(* CODESYS project SmiuUGP.project

Project tree, tasks and I/O mapping:
  CODESYS_Control_for_Raspberry_Pi : CODESYS Control for Raspberry Pi, 3S - Smart Software Solutions GmbH, version 3.5.7.10
    application Application
      libraries: Util, * (System); AlarmManager, * (Intern); Alarm Manager Interfaces, * (Intern); Standard, * (System); VisuDialogs, * (System)
      task MainTask (cyclic, interval t#50ms, priority 2, watchdog t#1000ms x 1) calls PLC_PRG, GPIO_HANDLER, AlarmChecker
      task VISU_TASK (cyclic, interval 100 ms, priority 30) calls VisuElems.Visu_Prg
      task AlarmManagerTask (cyclic, interval 50 ms, priority 31) calls AlarmManager.Alarm_Prg
      task BusTask (cyclic, interval t#20ms, priority 1, watchdog t#1000ms x 1) calls BusReinit
      program PLC_PRG [ST]
      image pool ImagePool
      program GPIO_HANDLER [ST]
      visualization/
        visualisation monitoring
        ups_s2/
          visualisation ups_s2_m1_state
          visualisation ups_s2_m1_params
          visualisation ups_s2
          visualisation ups_s2_m2_params
          visualisation ups_s2_m2_state
          visualisation ups_s2_m3_params
          visualisation ups_s2_m4_state
          visualisation ups_s2_m4_params
          visualisation ups_s2_m3_state
        visualisation test
        visualisation main
        visualisation info
        visualisation climate
        visualisation control
        visualisation alarm
        visualisation schrps
        visualisation shasn
        visualisation logs
        visualisation schrpa
        ups_s1/
          visualisation ups_s1
          visualisation ups_s1_m1_params
          visualisation ups_s1_m1_state
          visualisation ups_s1_m2_params
          visualisation ups_s1_m2_state
          visualisation ups_s1_m3_params
          visualisation ups_s1_m3_state
          visualisation ups_s1_m4_params
          visualisation ups_s1_m4_state
        ups_a1/
          visualisation ups_a1
          visualisation ups_a1_m1_params
          visualisation ups_a1_m1_state
          visualisation ups_a1_m2_params
          visualisation ups_a1_m2_state
        ups_a2/
          visualisation ups_a2
          visualisation ups_a2_m1_params
          visualisation ups_a2_m1_state
          visualisation ups_a2_m2_params
          visualisation ups_a2_m2_state
        visualisation climate_log
        visualisation more
      program InterviewState [ST]
      Alarm Configuration
        alarm class Error (priority 10, acknowledge REP)
        alarm class Warning (priority 30, acknowledge REP)
        alarm class Info (priority 100, acknowledge REP)
        AlarmStorage
        text list AlarmGroup
        alarm group AlarmGroup
            56 [Error]: Comparison Equal, ExpressionToCompare TRUE, Expression PLC_PRG.mpx_s2_4_alarm - "Авария ИБПС 2 модуль 4"
            46 [Error]: Comparison Equal, ExpressionToCompare TRUE, Expression PLC_PRG.mpx_a1_2_alarm - "Авария ИБПА 1 модуль 2"
            49 [Error]: Comparison Equal, ExpressionToCompare TRUE, Expression PLC_PRG.mpx_s1_1_alarm - "Авария ИБПС 1 модуль 1"
            51 [Error]: Comparison Equal, ExpressionToCompare TRUE, Expression PLC_PRG.mpx_s1_3_alarm - "Авария ИБПС 1 модуль 3"
            87 [Error]: Comparison Equal, ExpressionToCompare FALSE, Expression GPIO_HANDLER.IN_10 - "Отключен выходной автомат ИБПС 2"
            94 [Error]: Comparison Equal, ExpressionToCompare TRUE, Expression AlarmChecker.ups_a1_out_v_alarm - "Отсутствует напряжение на выходе ИБПА 1"
            54 [Error]: Comparison Equal, ExpressionToCompare TRUE, Expression PLC_PRG.mpx_s2_2_alarm - "Авария ИБПС 2 модуль 2"
            53 [Error]: Comparison Equal, ExpressionToCompare TRUE, Expression PLC_PRG.mpx_s2_1_alarm - "Авария ИБПС 2 модуль 1"
            92 [Error]: Comparison Equal, ExpressionToCompare TRUE, Expression AlarmChecker.ups_s1_out_v_alarm - "Отсутствует напряжение на выходе ИБПС 1"
            85 [Error]: Comparison Equal, ExpressionToCompare FALSE, Expression GPIO_HANDLER.IN_8 - "Отключен выходной автомат ИБПС 1"
            47 [Error]: Comparison Equal, ExpressionToCompare TRUE, Expression PLC_PRG.mpx_a2_1_alarm - "Авария ИБПА 2 модуль 1"
            90 [Error]: Comparison Equal, ExpressionToCompare TRUE, Expression AlarmChecker.ups_a1_in_v_alarm - "Отсутствует напряжение на входе ИБПА 1"
            52 [Error]: Comparison Equal, ExpressionToCompare TRUE, Expression PLC_PRG.mpx_s1_4_alarm - "Авария ИБПС 1 модуль 4"
            1 [Error]: Comparison Equal, ExpressionToCompare FALSE, Expression GPIO_HANDLER.IN_5 - "Отсутствует напряжение на резервном вводе ЩРПА"
            2 [Error]: Comparison Equal, ExpressionToCompare FALSE, Expression PLC_PRG.mv110_in_0_in_main_present - "Отсутствует напряжение на основном вводе ШАСН"
            6 [Error]: Comparison Equal, ExpressionToCompare FALSE, Expression PLC_PRG.mv110_in_2_bp_sn_present - "Отсутствует напряжение на шине БП ШАСН"
            4 [Error]: Comparison Equal, ExpressionToCompare TRUE, Expression PLC_PRG.mv110_in_7_gp1_u_fault - "Отсутствует напряжение на ГП 1 ЩРПС"
            5 [Error]: Comparison Equal, ExpressionToCompare TRUE, Expression PLC_PRG.mv110_in_8_gp2_u_fault - "Отсутствует напряжение на ГП 2 ЩРПС"
            93 [Error]: Comparison Equal, ExpressionToCompare TRUE, Expression AlarmChecker.ups_s2_out_v_alarm - "Отсутствует напряжение на выходе ИБПС 2"
            48 [Error]: Comparison Equal, ExpressionToCompare TRUE, Expression PLC_PRG.mpx_a2_2_alarm - "Авария ИБПА 2 модуль 2"
            45 [Error]: Comparison Equal, ExpressionToCompare TRUE, Expression PLC_PRG.mpx_a1_1_alarm - "Авария ИБПА 1 модуль 1"
            88 [Error]: Comparison Equal, ExpressionToCompare TRUE, Expression AlarmChecker.ups_s1_in_v_alarm - "Отсутствует напряжение на входе ИБПС 1"
            50 [Error]: Comparison Equal, ExpressionToCompare TRUE, Expression PLC_PRG.mpx_s1_2_alarm - "Авария ИБПС 1 модуль 2"
            95 [Error]: Comparison Equal, ExpressionToCompare TRUE, Expression AlarmChecker.ups_a2_out_v_alarm - "Отсутствует напряжение на выходе ИБПА 2"
            89 [Error]: Comparison Equal, ExpressionToCompare TRUE, Expression AlarmChecker.ups_s2_in_v_alarm - "Отсутствует напряжение на входе ИБПС 2"
            0 [Error]: Comparison Equal, ExpressionToCompare FALSE, Expression GPIO_HANDLER.IN_4 - "Отсутствует напряжение на основном вводе ЩРПА"
            91 [Error]: Comparison Equal, ExpressionToCompare TRUE, Expression AlarmChecker.ups_a2_in_v_alarm - "Отсутствует напряжение на входе ИБПА 2"
            55 [Error]: Comparison Equal, ExpressionToCompare TRUE, Expression PLC_PRG.mpx_s2_3_alarm - "Авария ИБПС 2 модуль 3"
            3 [Error]: Comparison Equal, ExpressionToCompare FALSE, Expression PLC_PRG.mv110_in_1_in_reserve_present - "Отсутствует напряжение на резервном вводе ШАСН"
            7 [Error]: Comparison Equal, ExpressionToCompare FALSE, Expression PLC_PRG.mv110_in_3_gp_sn_present - "Отсутствует напряжение на шине ГП ШАСН"
        text list ClimateGroup
        alarm group ClimateGroup
            1 [Info]: Comparison Equal, ExpressionToCompare TRUE, Expression PLC_PRG.climate_auto_state - "Автоматика включена"
            2 [Info]: Comparison Equal, ExpressionToCompare FALSE, Expression PLC_PRG.climate_heat_state - "Обогрев выключен"
            3 [Info]: Comparison Equal, ExpressionToCompare FALSE, Expression PLC_PRG.climate_auto_state - "Автоматика выключена"
            4 [Info]: Comparison Equal, ExpressionToCompare TRUE, Expression PLC_PRG.climate_zaslonka_state - "Заслонка открыта"
            5 [Info]: Comparison Equal, ExpressionToCompare FALSE, Expression PLC_PRG.climate_zaslonka_state - "Заслонка закрыта"
            11 [Info]: Comparison Equal, ExpressionToCompare FALSE, Expression PLC_PRG.climate_heat_door_state - "Обогрев дверей выключен"
            7 [Info]: Comparison Equal, ExpressionToCompare FALSE, Expression PLC_PRG.climate_vent_1_state - "Вентиляторы выключены"
            6 [Info]: Comparison Equal, ExpressionToCompare TRUE, Expression PLC_PRG.climate_vent_1_state - "Вентиляторы включены"
            8 [Info]: Comparison Equal, ExpressionToCompare TRUE, Expression PLC_PRG.climate_condition_1_state - "Кондиционеры включены"
            9 [Info]: Comparison Equal, ExpressionToCompare FALSE, Expression PLC_PRG.climate_condition_1_state - "Кондиционеры выключены"
            10 [Info]: Comparison Equal, ExpressionToCompare TRUE, Expression PLC_PRG.climate_heat_door_state - "Обогрев дверей включен"
            0 [Info]: Comparison Equal, ExpressionToCompare TRUE, Expression PLC_PRG.climate_heat_state - "Обогрев включен"
      program BusReinit [ST]
      program AlarmChecker [ST]
    SoftMotion General Axis Pool
    GPIOs_B_Pi2 : GPIOs B+/Pi2, 3S - Smart Software Solutions GmbH, version 1.1.1.10
        input  Application.GPIO_HANDLER.IN_10 : BOOL  // digital inputs (GPIO0..GPIO31).Bit5
        input  Application.GPIO_HANDLER.IN_12 : BOOL  // digital inputs (GPIO0..GPIO31).Bit6
        input  Application.GPIO_HANDLER.IN_9 : BOOL  // digital inputs (GPIO0..GPIO31).Bit7
        input  Application.GPIO_HANDLER.IN_8 : BOOL  // digital inputs (GPIO0..GPIO31).Bit8
        input  Application.GPIO_HANDLER.IN_3 : BOOL  // digital inputs (GPIO0..GPIO31).Bit10
        input  Application.GPIO_HANDLER.IN_11 : BOOL  // digital inputs (GPIO0..GPIO31).Bit12
        input  Application.GPIO_HANDLER.IN_1 : BOOL  // digital inputs (GPIO0..GPIO31).Bit13
        input  Application.GPIO_HANDLER.IN_6 : BOOL  // digital inputs (GPIO0..GPIO31).Bit18
        input  Application.GPIO_HANDLER.IN_7 : BOOL  // digital inputs (GPIO0..GPIO31).Bit21
        input  Application.GPIO_HANDLER.IN_5 : BOOL  // digital inputs (GPIO0..GPIO31).Bit23
        input  Application.GPIO_HANDLER.IN_4 : BOOL  // digital inputs (GPIO0..GPIO31).Bit24
        input  Application.GPIO_HANDLER.IN_2 : BOOL  // digital inputs (GPIO0..GPIO31).Bit25
        unmapped channels: digital inputs (GPIO0..GPIO31), digital outputs (GPIO0..GPIO31)
    Camera device
      <Empty>
    I²C
    SPI
    Onewire
    Ethernet : Ethernet, 3S - Smart Software Solutions GmbH, version 3.4.2.0
        settings: IPAddress = [192,168,10,200]; SubnetMask = [255,255,255,0]; GatewayAddress = [0,0,0,0]; NetworkInterfaceName = 'eth0'; NetworkInterfaceName = "eth0"
      Modbus_TCP_Master : Modbus TCP Master, 3S - Smart Software Solutions GmbH, version 3.5.4.0
          settings: AutoReconnect = TRUE
        MPX_S2_1 : Modbus TCP Slave, 3S - Smart Software Solutions GmbH, version 3.5.4.0
            settings: Unit-ID = 1; ResponseTimeout = 1500; IPAddress = [192, 168, 10, 108]; bypass_out.Function Code = 3; bypass_out.Read Offset = 16#0015; bypass_out.Read Length = 7; bypass_out.Write Offset = 0; bypass_out.Write Length = 0; bypass_out.Cycle Time = 300; output.Function Code = 3; output.Read Offset = 16#001F; output.Read Length = 13; output.Write Offset = 0; output.Write Length = 0; output.Cycle Time = 300; battery.Function Code = 3; battery.Read Offset = 16#002F; battery.Read Length = 7; battery.Write Offset = 0; battery.Write Length = 0; battery.Cycle Time = 300; states.Function Code = 3; states.Read Offset = 16#0000; states.Read Length = 2; states.Write Offset = 0; states.Write Length = 0; states.Cycle Time = 300; input.Function Code = 3; input.Read Offset = 16#000B; input.Read Length = 7; input.Write Offset = 0; input.Write Length = 0; input.Cycle Time = 300; temp.Function Code = 3; temp.Read Offset = 16#003D; temp.Read Length = 1; temp.Write Offset = 0; temp.Write Length = 0; temp.Cycle Time = 300; battery_test.Function Code = 6;
              battery_test.Read Offset = 0; battery_test.Read Length = 0; battery_test.Write Offset = 16#0070; battery_test.Write Length = 1; battery_test.Cycle Time = 100
            input  Application.PLC_PRG.mpx_s2_1_bypass_v_1 : WORD  // bypass_out.bypass_out
            input  Application.PLC_PRG.mpx_s2_1_bypass_v_2 : WORD  // bypass_out.bypass_out
            input  Application.PLC_PRG.mpx_s2_1_bypass_v_3 : WORD  // bypass_out.bypass_out
            input  Application.PLC_PRG.mpx_s2_1_bypass_freq : WORD  // bypass_out.bypass_out
            input  Application.PLC_PRG.mpx_s2_1_output_v_1 : WORD  // bypass_out.bypass_out
            input  Application.PLC_PRG.mpx_s2_1_output_v_2 : WORD  // bypass_out.bypass_out
            input  Application.PLC_PRG.mpx_s2_1_output_v_3 : WORD  // bypass_out.bypass_out
            input  Application.PLC_PRG.mpx_s2_1_output_i_1 : WORD  // output.output
            input  Application.PLC_PRG.mpx_s2_1_output_i_2 : WORD  // output.output
            input  Application.PLC_PRG.mpx_s2_1_output_i_3 : WORD  // output.output
            input  Application.PLC_PRG.mpx_s2_1_load_ph_1 : WORD  // output.output
            input  Application.PLC_PRG.mpx_s2_1_load_ph_2 : WORD  // output.output
            input  Application.PLC_PRG.mpx_s2_1_load_ph_3 : WORD  // output.output
            input  Application.PLC_PRG.mpx_s2_1_output_active_power_1 : WORD  // output.output
            input  Application.PLC_PRG.mpx_s2_1_output_active_power_2 : WORD  // output.output
            input  Application.PLC_PRG.mpx_s2_1_output_active_power_3 : WORD  // output.output
            input  Application.PLC_PRG.mpx_s2_1_output_freq : WORD  // output.output
            input  Application.PLC_PRG.mpx_s2_1_battery_voltage : WORD  // battery.battery
            input  Application.PLC_PRG.mpx_s2_1_battery_current : WORD  // battery.battery
            input  Application.PLC_PRG.mpx_s2_1_battery_capacity : WORD  // battery.battery
            input  Application.PLC_PRG.mpx_s2_1_battery_time : WORD  // battery.battery
            input  Application.PLC_PRG.mpx_s2_1_state_reg_1 : WORD  // states.states
            input  Application.PLC_PRG.mpx_s2_1_state_reg_2 : WORD  // states.states
            input  Application.PLC_PRG.mpx_s2_1_in_v_1 : WORD  // input.input
            input  Application.PLC_PRG.mpx_s2_1_in_v_2 : WORD  // input.input
            input  Application.PLC_PRG.mpx_s2_1_in_v_3 : WORD  // input.input
            input  Application.PLC_PRG.mpx_s2_1_in_freq : WORD  // input.input
            input  Application.PLC_PRG.mpx_s2_1_temp : WORD  // temp.temp
            output Application.PLC_PRG.mpx_s2_test_battery_start : BIT  // battery_test
            output Application.PLC_PRG.mpx_test_battery_command : ARRAY[0..0] OF WORD  // battery_test
            unmapped channels: bypass_out, output, battery, states, input, temp
        MPX_S2_4 : Modbus TCP Slave, 3S - Smart Software Solutions GmbH, version 3.5.4.0
            settings: Unit-ID = 1; ResponseTimeout = 1500; IPAddress = [192, 168, 10, 105]; bypass_out.Function Code = 3; bypass_out.Read Offset = 16#0015; bypass_out.Read Length = 7; bypass_out.Write Offset = 0; bypass_out.Write Length = 0; bypass_out.Cycle Time = 300; output.Function Code = 3; output.Read Offset = 16#001F; output.Read Length = 13; output.Write Offset = 0; output.Write Length = 0; output.Cycle Time = 300; battery.Function Code = 3; battery.Read Offset = 16#002F; battery.Read Length = 7; battery.Write Offset = 0; battery.Write Length = 0; battery.Cycle Time = 300; states.Function Code = 3; states.Read Offset = 16#0000; states.Read Length = 2; states.Write Offset = 0; states.Write Length = 0; states.Cycle Time = 300; input.Function Code = 3; input.Read Offset = 16#000B; input.Read Length = 7; input.Write Offset = 0; input.Write Length = 0; input.Cycle Time = 300; temp.Function Code = 3; temp.Read Offset = 16#003D; temp.Read Length = 1; temp.Write Offset = 0; temp.Write Length = 0; temp.Cycle Time = 300; battery_test.Function Code = 6;
              battery_test.Read Offset = 0; battery_test.Read Length = 0; battery_test.Write Offset = 16#0070; battery_test.Write Length = 1; battery_test.Cycle Time = 100
            input  Application.PLC_PRG.mpx_s2_4_bypass_v_1 : WORD  // bypass_out.bypass_out
            input  Application.PLC_PRG.mpx_s2_4_bypass_v_2 : WORD  // bypass_out.bypass_out
            input  Application.PLC_PRG.mpx_s2_4_bypass_v_3 : WORD  // bypass_out.bypass_out
            input  Application.PLC_PRG.mpx_s2_4_bypass_freq : WORD  // bypass_out.bypass_out
            input  Application.PLC_PRG.mpx_s2_4_output_v_1 : WORD  // bypass_out.bypass_out
            input  Application.PLC_PRG.mpx_s2_4_output_v_2 : WORD  // bypass_out.bypass_out
            input  Application.PLC_PRG.mpx_s2_4_output_v_3 : WORD  // bypass_out.bypass_out
            input  Application.PLC_PRG.mpx_s2_4_output_i_1 : WORD  // output.output
            input  Application.PLC_PRG.mpx_s2_4_output_i_2 : WORD  // output.output
            input  Application.PLC_PRG.mpx_s2_4_output_i_3 : WORD  // output.output
            input  Application.PLC_PRG.mpx_s2_4_load_ph_1 : WORD  // output.output
            input  Application.PLC_PRG.mpx_s2_4_load_ph_2 : WORD  // output.output
            input  Application.PLC_PRG.mpx_s2_4_load_ph_3 : WORD  // output.output
            input  Application.PLC_PRG.mpx_s2_4_output_active_power_1 : WORD  // output.output
            input  Application.PLC_PRG.mpx_s2_4_output_active_power_2 : WORD  // output.output
            input  Application.PLC_PRG.mpx_s2_4_output_active_power_3 : WORD  // output.output
            input  Application.PLC_PRG.mpx_s2_4_output_freq : WORD  // output.output
            input  Application.PLC_PRG.mpx_s2_4_battery_voltage : WORD  // battery.battery
            input  Application.PLC_PRG.mpx_s2_4_battery_current : WORD  // battery.battery
            input  Application.PLC_PRG.mpx_s2_4_battery_capacity : WORD  // battery.battery
            input  Application.PLC_PRG.mpx_s2_4_battery_time : WORD  // battery.battery
            input  Application.PLC_PRG.mpx_s2_4_state_reg_1 : WORD  // states.states
            input  Application.PLC_PRG.mpx_s2_4_state_reg_2 : WORD  // states.states
            input  Application.PLC_PRG.mpx_s2_4_in_v_1 : WORD  // input.input
            input  Application.PLC_PRG.mpx_s2_4_in_v_2 : WORD  // input.input
            input  Application.PLC_PRG.mpx_s2_4_in_v_3 : WORD  // input.input
            input  Application.PLC_PRG.mpx_s2_4_in_freq : WORD  // input.input
            input  Application.PLC_PRG.mpx_s2_4_temp : WORD  // temp.temp
            output Application.PLC_PRG.mpx_s2_test_battery_start : BIT  // battery_test
            output Application.PLC_PRG.mpx_test_battery_command : ARRAY[0..0] OF WORD  // battery_test
            unmapped channels: bypass_out, output, battery, states, input, temp
        MPX_S2_3 : Modbus TCP Slave, 3S - Smart Software Solutions GmbH, version 3.5.4.0
            settings: Unit-ID = 1; ResponseTimeout = 1500; IPAddress = [192, 168, 10, 106]; bypass_out.Function Code = 3; bypass_out.Read Offset = 16#0015; bypass_out.Read Length = 7; bypass_out.Write Offset = 0; bypass_out.Write Length = 0; bypass_out.Cycle Time = 300; output.Function Code = 3; output.Read Offset = 16#001F; output.Read Length = 13; output.Write Offset = 0; output.Write Length = 0; output.Cycle Time = 300; battery.Function Code = 3; battery.Read Offset = 16#002F; battery.Read Length = 7; battery.Write Offset = 0; battery.Write Length = 0; battery.Cycle Time = 300; states.Function Code = 3; states.Read Offset = 16#0000; states.Read Length = 2; states.Write Offset = 0; states.Write Length = 0; states.Cycle Time = 300; input.Function Code = 3; input.Read Offset = 16#000B; input.Read Length = 7; input.Write Offset = 0; input.Write Length = 0; input.Cycle Time = 300; temp.Function Code = 3; temp.Read Offset = 16#003D; temp.Read Length = 1; temp.Write Offset = 0; temp.Write Length = 0; temp.Cycle Time = 300; battery_test.Function Code = 6;
              battery_test.Read Offset = 0; battery_test.Read Length = 0; battery_test.Write Offset = 16#0070; battery_test.Write Length = 1; battery_test.Cycle Time = 100
            input  Application.PLC_PRG.mpx_s2_3_bypass_v_1 : WORD  // bypass_out.bypass_out
            input  Application.PLC_PRG.mpx_s2_3_bypass_v_2 : WORD  // bypass_out.bypass_out
            input  Application.PLC_PRG.mpx_s2_3_bypass_v_3 : WORD  // bypass_out.bypass_out
            input  Application.PLC_PRG.mpx_s2_3_bypass_freq : WORD  // bypass_out.bypass_out
            input  Application.PLC_PRG.mpx_s2_3_output_v_1 : WORD  // bypass_out.bypass_out
            input  Application.PLC_PRG.mpx_s2_3_output_v_2 : WORD  // bypass_out.bypass_out
            input  Application.PLC_PRG.mpx_s2_3_output_v_3 : WORD  // bypass_out.bypass_out
            input  Application.PLC_PRG.mpx_s2_3_output_i_1 : WORD  // output.output
            input  Application.PLC_PRG.mpx_s2_3_output_i_2 : WORD  // output.output
            input  Application.PLC_PRG.mpx_s2_3_output_i_3 : WORD  // output.output
            input  Application.PLC_PRG.mpx_s2_3_load_ph_1 : WORD  // output.output
            input  Application.PLC_PRG.mpx_s2_3_load_ph_2 : WORD  // output.output
            input  Application.PLC_PRG.mpx_s2_3_load_ph_3 : WORD  // output.output
            input  Application.PLC_PRG.mpx_s2_3_output_active_power_1 : WORD  // output.output
            input  Application.PLC_PRG.mpx_s2_3_output_active_power_2 : WORD  // output.output
            input  Application.PLC_PRG.mpx_s2_3_output_active_power_3 : WORD  // output.output
            input  Application.PLC_PRG.mpx_s2_3_output_freq : WORD  // output.output
            input  Application.PLC_PRG.mpx_s2_3_battery_voltage : WORD  // battery.battery
            input  Application.PLC_PRG.mpx_s2_3_battery_current : WORD  // battery.battery
            input  Application.PLC_PRG.mpx_s2_3_battery_capacity : WORD  // battery.battery
            input  Application.PLC_PRG.mpx_s2_3_battery_time : WORD  // battery.battery
            input  Application.PLC_PRG.mpx_s2_3_state_reg_1 : WORD  // states.states
            input  Application.PLC_PRG.mpx_s2_3_state_reg_2 : WORD  // states.states
            input  Application.PLC_PRG.mpx_s2_3_in_v_1 : WORD  // input.input
            input  Application.PLC_PRG.mpx_s2_3_in_v_2 : WORD  // input.input
            input  Application.PLC_PRG.mpx_s2_3_in_v_3 : WORD  // input.input
            input  Application.PLC_PRG.mpx_s2_3_in_freq : WORD  // input.input
            input  Application.PLC_PRG.mpx_s2_3_temp : WORD  // temp.temp
            output Application.PLC_PRG.mpx_s2_test_battery_start : BIT  // battery_test
            output Application.PLC_PRG.mpx_test_battery_command : ARRAY[0..0] OF WORD  // battery_test
            unmapped channels: bypass_out, output, battery, states, input, temp
        MPX_S2_2 : Modbus TCP Slave, 3S - Smart Software Solutions GmbH, version 3.5.4.0
            settings: Unit-ID = 1; ResponseTimeout = 1500; IPAddress = [192, 168, 10, 107]; bypass_out.Function Code = 3; bypass_out.Read Offset = 16#0015; bypass_out.Read Length = 7; bypass_out.Write Offset = 0; bypass_out.Write Length = 0; bypass_out.Cycle Time = 300; output.Function Code = 3; output.Read Offset = 16#001F; output.Read Length = 13; output.Write Offset = 0; output.Write Length = 0; output.Cycle Time = 300; battery.Function Code = 3; battery.Read Offset = 16#002F; battery.Read Length = 7; battery.Write Offset = 0; battery.Write Length = 0; battery.Cycle Time = 300; states.Function Code = 3; states.Read Offset = 16#0000; states.Read Length = 2; states.Write Offset = 0; states.Write Length = 0; states.Cycle Time = 300; input.Function Code = 3; input.Read Offset = 16#000B; input.Read Length = 7; input.Write Offset = 0; input.Write Length = 0; input.Cycle Time = 300; temp.Function Code = 3; temp.Read Offset = 16#003D; temp.Read Length = 1; temp.Write Offset = 0; temp.Write Length = 0; temp.Cycle Time = 300; battery_test.Function Code = 6;
              battery_test.Read Offset = 0; battery_test.Read Length = 0; battery_test.Write Offset = 16#0070; battery_test.Write Length = 1; battery_test.Cycle Time = 100
            input  Application.PLC_PRG.mpx_s2_2_bypass_v_1 : WORD  // bypass_out.bypass_out
            input  Application.PLC_PRG.mpx_s2_2_bypass_v_2 : WORD  // bypass_out.bypass_out
            input  Application.PLC_PRG.mpx_s2_2_bypass_v_3 : WORD  // bypass_out.bypass_out
            input  Application.PLC_PRG.mpx_s2_2_bypass_freq : WORD  // bypass_out.bypass_out
            input  Application.PLC_PRG.mpx_s2_2_output_v_1 : WORD  // bypass_out.bypass_out
            input  Application.PLC_PRG.mpx_s2_2_output_v_2 : WORD  // bypass_out.bypass_out
            input  Application.PLC_PRG.mpx_s2_2_output_v_3 : WORD  // bypass_out.bypass_out
            input  Application.PLC_PRG.mpx_s2_2_output_i_1 : WORD  // output.output
            input  Application.PLC_PRG.mpx_s2_2_output_i_2 : WORD  // output.output
            input  Application.PLC_PRG.mpx_s2_2_output_i_3 : WORD  // output.output
            input  Application.PLC_PRG.mpx_s2_2_load_ph_1 : WORD  // output.output
            input  Application.PLC_PRG.mpx_s2_2_load_ph_2 : WORD  // output.output
            input  Application.PLC_PRG.mpx_s2_2_load_ph_3 : WORD  // output.output
            input  Application.PLC_PRG.mpx_s2_2_output_active_power_1 : WORD  // output.output
            input  Application.PLC_PRG.mpx_s2_2_output_active_power_2 : WORD  // output.output
            input  Application.PLC_PRG.mpx_s2_2_output_active_power_3 : WORD  // output.output
            input  Application.PLC_PRG.mpx_s2_2_output_freq : WORD  // output.output
            input  Application.PLC_PRG.mpx_s2_2_battery_voltage : WORD  // battery.battery
            input  Application.PLC_PRG.mpx_s2_2_battery_current : WORD  // battery.battery
            input  Application.PLC_PRG.mpx_s2_2_battery_capacity : WORD  // battery.battery
            input  Application.PLC_PRG.mpx_s2_2_battery_time : WORD  // battery.battery
            input  Application.PLC_PRG.mpx_s2_2_state_reg_1 : WORD  // states.states
            input  Application.PLC_PRG.mpx_s2_2_state_reg_2 : WORD  // states.states
            input  Application.PLC_PRG.mpx_s2_2_in_v_1 : WORD  // input.input
            input  Application.PLC_PRG.mpx_s2_2_in_v_2 : WORD  // input.input
            input  Application.PLC_PRG.mpx_s2_2_in_v_3 : WORD  // input.input
            input  Application.PLC_PRG.mpx_s2_2_in_freq : WORD  // input.input
            input  Application.PLC_PRG.mpx_s2_2_temp : WORD  // temp.temp
            output Application.PLC_PRG.mpx_s2_test_battery_start : BIT  // battery_test
            output Application.PLC_PRG.mpx_test_battery_command : ARRAY[0..0] OF WORD  // battery_test
            unmapped channels: bypass_out, output, battery, states, input, temp
        MPX_S1_1 : Modbus TCP Slave, 3S - Smart Software Solutions GmbH, version 3.5.4.0
            settings: Unit-ID = 1; ResponseTimeout = 1500; IPAddress = [192, 168, 10, 104]; bypass_out.Function Code = 3; bypass_out.Read Offset = 16#0015; bypass_out.Read Length = 7; bypass_out.Write Offset = 0; bypass_out.Write Length = 0; bypass_out.Cycle Time = 300; output.Function Code = 3; output.Read Offset = 16#001F; output.Read Length = 13; output.Write Offset = 0; output.Write Length = 0; output.Cycle Time = 300; battery.Function Code = 3; battery.Read Offset = 16#002F; battery.Read Length = 7; battery.Write Offset = 0; battery.Write Length = 0; battery.Cycle Time = 300; states.Function Code = 3; states.Read Offset = 16#0000; states.Read Length = 2; states.Write Offset = 0; states.Write Length = 0; states.Cycle Time = 300; input.Function Code = 3; input.Read Offset = 16#000B; input.Read Length = 7; input.Write Offset = 0; input.Write Length = 0; input.Cycle Time = 300; temp.Function Code = 3; temp.Read Offset = 16#003D; temp.Read Length = 1; temp.Write Offset = 0; temp.Write Length = 0; temp.Cycle Time = 300; battery_test.Function Code = 6;
              battery_test.Read Offset = 0; battery_test.Read Length = 0; battery_test.Write Offset = 16#0070; battery_test.Write Length = 1; battery_test.Cycle Time = 100
            input  Application.PLC_PRG.mpx_s1_1_bypass_v_1 : WORD  // bypass_out.bypass_out
            input  Application.PLC_PRG.mpx_s1_1_bypass_v_2 : WORD  // bypass_out.bypass_out
            input  Application.PLC_PRG.mpx_s1_1_bypass_v_3 : WORD  // bypass_out.bypass_out
            input  Application.PLC_PRG.mpx_s1_1_bypass_freq : WORD  // bypass_out.bypass_out
            input  Application.PLC_PRG.mpx_s1_1_output_v_1 : WORD  // bypass_out.bypass_out
            input  Application.PLC_PRG.mpx_s1_1_output_v_2 : WORD  // bypass_out.bypass_out
            input  Application.PLC_PRG.mpx_s1_1_output_v_3 : WORD  // bypass_out.bypass_out
            input  Application.PLC_PRG.mpx_s1_1_output_i_1 : WORD  // output.output
            input  Application.PLC_PRG.mpx_s1_1_output_i_2 : WORD  // output.output
            input  Application.PLC_PRG.mpx_s1_1_output_i_3 : WORD  // output.output
            input  Application.PLC_PRG.mpx_s1_1_load_ph_1 : WORD  // output.output
            input  Application.PLC_PRG.mpx_s1_1_load_ph_2 : WORD  // output.output
            input  Application.PLC_PRG.mpx_s1_1_load_ph_3 : WORD  // output.output
            input  Application.PLC_PRG.mpx_s1_1_output_active_power_1 : WORD  // output.output
            input  Application.PLC_PRG.mpx_s1_1_output_active_power_2 : WORD  // output.output
            input  Application.PLC_PRG.mpx_s1_1_output_active_power_3 : WORD  // output.output
            input  Application.PLC_PRG.mpx_s1_1_output_freq : WORD  // output.output
            input  Application.PLC_PRG.mpx_s1_1_battery_voltage : WORD  // battery.battery
            input  Application.PLC_PRG.mpx_s1_1_battery_current : WORD  // battery.battery
            input  Application.PLC_PRG.mpx_s1_1_battery_capacity : WORD  // battery.battery
            input  Application.PLC_PRG.mpx_s1_1_battery_time : WORD  // battery.battery
            input  Application.PLC_PRG.mpx_s1_1_state_reg_1 : WORD  // states.states
            input  Application.PLC_PRG.mpx_s1_1_state_reg_2 : WORD  // states.states
            input  Application.PLC_PRG.mpx_s1_1_in_v_1 : WORD  // input.input
            input  Application.PLC_PRG.mpx_s1_1_in_v_2 : WORD  // input.input
            input  Application.PLC_PRG.mpx_s1_1_in_v_3 : WORD  // input.input
            input  Application.PLC_PRG.mpx_s1_1_in_freq : WORD  // input.input
            input  Application.PLC_PRG.mpx_s1_1_temp : WORD  // temp.temp
            output Application.PLC_PRG.mpx_s1_test_battery_start : BIT  // battery_test
            output Application.PLC_PRG.mpx_test_battery_command : ARRAY[0..0] OF WORD  // battery_test
            unmapped channels: bypass_out, output, battery, states, input, temp
        MPX_S1_2 : Modbus TCP Slave, 3S - Smart Software Solutions GmbH, version 3.5.4.0
            settings: Unit-ID = 1; ResponseTimeout = 1500; IPAddress = [192, 168, 10, 103]; bypass_out.Function Code = 3; bypass_out.Read Offset = 16#0015; bypass_out.Read Length = 7; bypass_out.Write Offset = 0; bypass_out.Write Length = 0; bypass_out.Cycle Time = 300; output.Function Code = 3; output.Read Offset = 16#001F; output.Read Length = 13; output.Write Offset = 0; output.Write Length = 0; output.Cycle Time = 300; battery.Function Code = 3; battery.Read Offset = 16#002F; battery.Read Length = 7; battery.Write Offset = 0; battery.Write Length = 0; battery.Cycle Time = 300; states.Function Code = 3; states.Read Offset = 16#0000; states.Read Length = 2; states.Write Offset = 0; states.Write Length = 0; states.Cycle Time = 300; input.Function Code = 3; input.Read Offset = 16#000B; input.Read Length = 7; input.Write Offset = 0; input.Write Length = 0; input.Cycle Time = 300; temp.Function Code = 3; temp.Read Offset = 16#003D; temp.Read Length = 1; temp.Write Offset = 0; temp.Write Length = 0; temp.Cycle Time = 300; battery_test.Function Code = 6;
              battery_test.Read Offset = 0; battery_test.Read Length = 0; battery_test.Write Offset = 16#0070; battery_test.Write Length = 1; battery_test.Cycle Time = 100
            input  Application.PLC_PRG.mpx_s1_2_bypass_v_1 : WORD  // bypass_out.bypass_out
            input  Application.PLC_PRG.mpx_s1_2_bypass_v_2 : WORD  // bypass_out.bypass_out
            input  Application.PLC_PRG.mpx_s1_2_bypass_v_3 : WORD  // bypass_out.bypass_out
            input  Application.PLC_PRG.mpx_s1_2_bypass_freq : WORD  // bypass_out.bypass_out
            input  Application.PLC_PRG.mpx_s1_2_output_v_1 : WORD  // bypass_out.bypass_out
            input  Application.PLC_PRG.mpx_s1_2_output_v_2 : WORD  // bypass_out.bypass_out
            input  Application.PLC_PRG.mpx_s1_2_output_v_3 : WORD  // bypass_out.bypass_out
            input  Application.PLC_PRG.mpx_s1_2_output_i_1 : WORD  // output.output
            input  Application.PLC_PRG.mpx_s1_2_output_i_2 : WORD  // output.output
            input  Application.PLC_PRG.mpx_s1_2_output_i_3 : WORD  // output.output
            input  Application.PLC_PRG.mpx_s1_2_load_ph_1 : WORD  // output.output
            input  Application.PLC_PRG.mpx_s1_2_load_ph_2 : WORD  // output.output
            input  Application.PLC_PRG.mpx_s1_2_load_ph_3 : WORD  // output.output
            input  Application.PLC_PRG.mpx_s1_2_output_active_power_1 : WORD  // output.output
            input  Application.PLC_PRG.mpx_s1_2_output_active_power_2 : WORD  // output.output
            input  Application.PLC_PRG.mpx_s1_2_output_active_power_3 : WORD  // output.output
            input  Application.PLC_PRG.mpx_s1_2_output_freq : WORD  // output.output
            input  Application.PLC_PRG.mpx_s1_2_battery_voltage : WORD  // battery.battery
            input  Application.PLC_PRG.mpx_s1_2_battery_current : WORD  // battery.battery
            input  Application.PLC_PRG.mpx_s1_2_battery_capacity : WORD  // battery.battery
            input  Application.PLC_PRG.mpx_s1_2_battery_time : WORD  // battery.battery
            input  Application.PLC_PRG.mpx_s1_2_state_reg_1 : WORD  // states.states
            input  Application.PLC_PRG.mpx_s1_2_state_reg_2 : WORD  // states.states
            input  Application.PLC_PRG.mpx_s1_2_in_v_1 : WORD  // input.input
            input  Application.PLC_PRG.mpx_s1_2_in_v_2 : WORD  // input.input
            input  Application.PLC_PRG.mpx_s1_2_in_v_3 : WORD  // input.input
            input  Application.PLC_PRG.mpx_s1_2_in_freq : WORD  // input.input
            input  Application.PLC_PRG.mpx_s1_2_temp : WORD  // temp.temp
            output Application.PLC_PRG.mpx_s1_test_battery_start : BIT  // battery_test
            output Application.PLC_PRG.mpx_test_battery_command : ARRAY[0..0] OF WORD  // battery_test
            unmapped channels: bypass_out, output, battery, states, input, temp
        MPX_S1_3 : Modbus TCP Slave, 3S - Smart Software Solutions GmbH, version 3.5.4.0
            settings: Unit-ID = 1; ResponseTimeout = 1500; IPAddress = [192, 168, 10, 102]; bypass_out.Function Code = 3; bypass_out.Read Offset = 16#0015; bypass_out.Read Length = 7; bypass_out.Write Offset = 0; bypass_out.Write Length = 0; bypass_out.Cycle Time = 300; output.Function Code = 3; output.Read Offset = 16#001F; output.Read Length = 13; output.Write Offset = 0; output.Write Length = 0; output.Cycle Time = 300; battery.Function Code = 3; battery.Read Offset = 16#002F; battery.Read Length = 7; battery.Write Offset = 0; battery.Write Length = 0; battery.Cycle Time = 300; states.Function Code = 3; states.Read Offset = 16#0000; states.Read Length = 2; states.Write Offset = 0; states.Write Length = 0; states.Cycle Time = 300; input.Function Code = 3; input.Read Offset = 16#000B; input.Read Length = 7; input.Write Offset = 0; input.Write Length = 0; input.Cycle Time = 300; temp.Function Code = 3; temp.Read Offset = 16#003D; temp.Read Length = 1; temp.Write Offset = 0; temp.Write Length = 0; temp.Cycle Time = 300; battery_test.Function Code = 6;
              battery_test.Read Offset = 0; battery_test.Read Length = 0; battery_test.Write Offset = 16#0070; battery_test.Write Length = 1; battery_test.Cycle Time = 100
            input  Application.PLC_PRG.mpx_s1_3_bypass_v_1 : WORD  // bypass_out.bypass_out
            input  Application.PLC_PRG.mpx_s1_3_bypass_v_2 : WORD  // bypass_out.bypass_out
            input  Application.PLC_PRG.mpx_s1_3_bypass_v_3 : WORD  // bypass_out.bypass_out
            input  Application.PLC_PRG.mpx_s1_3_bypass_freq : WORD  // bypass_out.bypass_out
            input  Application.PLC_PRG.mpx_s1_3_output_v_1 : WORD  // bypass_out.bypass_out
            input  Application.PLC_PRG.mpx_s1_3_output_v_2 : WORD  // bypass_out.bypass_out
            input  Application.PLC_PRG.mpx_s1_3_output_v_3 : WORD  // bypass_out.bypass_out
            input  Application.PLC_PRG.mpx_s1_3_output_i_1 : WORD  // output.output
            input  Application.PLC_PRG.mpx_s1_3_output_i_2 : WORD  // output.output
            input  Application.PLC_PRG.mpx_s1_3_output_i_3 : WORD  // output.output
            input  Application.PLC_PRG.mpx_s1_3_load_ph_1 : WORD  // output.output
            input  Application.PLC_PRG.mpx_s1_3_load_ph_2 : WORD  // output.output
            input  Application.PLC_PRG.mpx_s1_3_load_ph_3 : WORD  // output.output
            input  Application.PLC_PRG.mpx_s1_3_output_active_power_1 : WORD  // output.output
            input  Application.PLC_PRG.mpx_s1_3_output_active_power_2 : WORD  // output.output
            input  Application.PLC_PRG.mpx_s1_3_output_active_power_3 : WORD  // output.output
            input  Application.PLC_PRG.mpx_s1_3_output_freq : WORD  // output.output
            input  Application.PLC_PRG.mpx_s1_3_battery_voltage : WORD  // battery.battery
            input  Application.PLC_PRG.mpx_s1_3_battery_current : WORD  // battery.battery
            input  Application.PLC_PRG.mpx_s1_3_battery_capacity : WORD  // battery.battery
            input  Application.PLC_PRG.mpx_s1_3_battery_time : WORD  // battery.battery
            input  Application.PLC_PRG.mpx_s1_3_state_reg_1 : WORD  // states.states
            input  Application.PLC_PRG.mpx_s1_3_state_reg_2 : WORD  // states.states
            input  Application.PLC_PRG.mpx_s1_3_in_v_1 : WORD  // input.input
            input  Application.PLC_PRG.mpx_s1_3_in_v_2 : WORD  // input.input
            input  Application.PLC_PRG.mpx_s1_3_in_v_3 : WORD  // input.input
            input  Application.PLC_PRG.mpx_s1_3_in_freq : WORD  // input.input
            input  Application.PLC_PRG.mpx_s1_3_temp : WORD  // temp.temp
            output Application.PLC_PRG.mpx_s1_test_battery_start : BIT  // battery_test
            output Application.PLC_PRG.mpx_test_battery_command : ARRAY[0..0] OF WORD  // battery_test
            unmapped channels: bypass_out, output, battery, states, input, temp
        MPX_S1_4 : Modbus TCP Slave, 3S - Smart Software Solutions GmbH, version 3.5.4.0
            settings: Unit-ID = 1; ResponseTimeout = 1500; IPAddress = [192, 168, 10, 101]; bypass_out.Function Code = 3; bypass_out.Read Offset = 16#0015; bypass_out.Read Length = 7; bypass_out.Write Offset = 0; bypass_out.Write Length = 0; bypass_out.Cycle Time = 300; output.Function Code = 3; output.Read Offset = 16#001F; output.Read Length = 13; output.Write Offset = 0; output.Write Length = 0; output.Cycle Time = 300; battery.Function Code = 3; battery.Read Offset = 16#002F; battery.Read Length = 7; battery.Write Offset = 0; battery.Write Length = 0; battery.Cycle Time = 300; states.Function Code = 3; states.Read Offset = 16#0000; states.Read Length = 2; states.Write Offset = 0; states.Write Length = 0; states.Cycle Time = 300; input.Function Code = 3; input.Read Offset = 16#000B; input.Read Length = 7; input.Write Offset = 0; input.Write Length = 0; input.Cycle Time = 300; temp.Function Code = 3; temp.Read Offset = 16#003D; temp.Read Length = 1; temp.Write Offset = 0; temp.Write Length = 0; temp.Cycle Time = 300; battery_test.Function Code = 6;
              battery_test.Read Offset = 0; battery_test.Read Length = 0; battery_test.Write Offset = 16#0070; battery_test.Write Length = 1; battery_test.Cycle Time = 100
            input  Application.PLC_PRG.mpx_s1_4_bypass_v_1 : WORD  // bypass_out.bypass_out
            input  Application.PLC_PRG.mpx_s1_4_bypass_v_2 : WORD  // bypass_out.bypass_out
            input  Application.PLC_PRG.mpx_s1_4_bypass_v_3 : WORD  // bypass_out.bypass_out
            input  Application.PLC_PRG.mpx_s1_4_bypass_freq : WORD  // bypass_out.bypass_out
            input  Application.PLC_PRG.mpx_s1_4_output_v_1 : WORD  // bypass_out.bypass_out
            input  Application.PLC_PRG.mpx_s1_4_output_v_2 : WORD  // bypass_out.bypass_out
            input  Application.PLC_PRG.mpx_s1_4_output_v_3 : WORD  // bypass_out.bypass_out
            input  Application.PLC_PRG.mpx_s1_4_output_i_1 : WORD  // output.output
            input  Application.PLC_PRG.mpx_s1_4_output_i_2 : WORD  // output.output
            input  Application.PLC_PRG.mpx_s1_4_output_i_3 : WORD  // output.output
            input  Application.PLC_PRG.mpx_s1_4_load_ph_1 : WORD  // output.output
            input  Application.PLC_PRG.mpx_s1_4_load_ph_2 : WORD  // output.output
            input  Application.PLC_PRG.mpx_s1_4_load_ph_3 : WORD  // output.output
            input  Application.PLC_PRG.mpx_s1_4_output_active_power_1 : WORD  // output.output
            input  Application.PLC_PRG.mpx_s1_4_output_active_power_2 : WORD  // output.output
            input  Application.PLC_PRG.mpx_s1_4_output_active_power_3 : WORD  // output.output
            input  Application.PLC_PRG.mpx_s1_4_output_freq : WORD  // output.output
            input  Application.PLC_PRG.mpx_s1_4_battery_voltage : WORD  // battery.battery
            input  Application.PLC_PRG.mpx_s1_4_battery_current : WORD  // battery.battery
            input  Application.PLC_PRG.mpx_s1_4_battery_capacity : WORD  // battery.battery
            input  Application.PLC_PRG.mpx_s1_4_battery_time : WORD  // battery.battery
            input  Application.PLC_PRG.mpx_s1_4_state_reg_1 : WORD  // states.states
            input  Application.PLC_PRG.mpx_s1_4_state_reg_2 : WORD  // states.states
            input  Application.PLC_PRG.mpx_s1_4_in_v_1 : WORD  // input.input
            input  Application.PLC_PRG.mpx_s1_4_in_v_2 : WORD  // input.input
            input  Application.PLC_PRG.mpx_s1_4_in_v_3 : WORD  // input.input
            input  Application.PLC_PRG.mpx_s1_4_in_freq : WORD  // input.input
            input  Application.PLC_PRG.mpx_s1_4_temp : WORD  // temp.temp
            output Application.PLC_PRG.mpx_s1_test_battery_start : BIT  // battery_test
            output Application.PLC_PRG.mpx_test_battery_command : ARRAY[0..0] OF WORD  // battery_test
            unmapped channels: bypass_out, output, battery, states, input, temp
        MPX_A1_1 : Modbus TCP Slave, 3S - Smart Software Solutions GmbH, version 3.5.4.0
            settings: Unit-ID = 1; ResponseTimeout = 1500; IPAddress = [192, 168, 10, 112]; bypass_out.Function Code = 3; bypass_out.Read Offset = 16#0015; bypass_out.Read Length = 7; bypass_out.Write Offset = 0; bypass_out.Write Length = 0; bypass_out.Cycle Time = 300; output.Function Code = 3; output.Read Offset = 16#001F; output.Read Length = 13; output.Write Offset = 0; output.Write Length = 0; output.Cycle Time = 300; battery.Function Code = 3; battery.Read Offset = 16#002F; battery.Read Length = 7; battery.Write Offset = 0; battery.Write Length = 0; battery.Cycle Time = 300; states.Function Code = 3; states.Read Offset = 16#0000; states.Read Length = 2; states.Write Offset = 0; states.Write Length = 0; states.Cycle Time = 300; input.Function Code = 3; input.Read Offset = 16#000B; input.Read Length = 7; input.Write Offset = 0; input.Write Length = 0; input.Cycle Time = 300; temp.Function Code = 3; temp.Read Offset = 16#003D; temp.Read Length = 1; temp.Write Offset = 0; temp.Write Length = 0; temp.Cycle Time = 300; battery_test.Function Code = 6;
              battery_test.Read Offset = 0; battery_test.Read Length = 0; battery_test.Write Offset = 16#0070; battery_test.Write Length = 1; battery_test.Cycle Time = 100
            input  Application.PLC_PRG.mpx_a1_1_bypass_v_1 : WORD  // bypass_out.bypass_out
            input  Application.PLC_PRG.mpx_a1_1_bypass_freq : WORD  // bypass_out.bypass_out
            input  Application.PLC_PRG.mpx_a1_1_output_v_1 : WORD  // bypass_out.bypass_out
            input  Application.PLC_PRG.mpx_a1_1_output_i_1 : WORD  // output.output
            input  Application.PLC_PRG.mpx_a1_1_load_ph_1 : WORD  // output.output
            input  Application.PLC_PRG.mpx_a1_1_output_active_power_1 : WORD  // output.output
            input  Application.PLC_PRG.mpx_a1_1_output_freq : WORD  // output.output
            input  Application.PLC_PRG.mpx_a1_1_battery_voltage : WORD  // battery.battery
            input  Application.PLC_PRG.mpx_a1_1_battery_current : WORD  // battery.battery
            input  Application.PLC_PRG.mpx_a1_1_battery_capacity : WORD  // battery.battery
            input  Application.PLC_PRG.mpx_a1_1_battery_time : WORD  // battery.battery
            input  Application.PLC_PRG.mpx_a1_1_state_reg_1 : WORD  // states.states
            input  Application.PLC_PRG.mpx_a1_1_state_reg_2 : WORD  // states.states
            input  Application.PLC_PRG.mpx_a1_1_in_v_1 : WORD  // input.input
            input  Application.PLC_PRG.mpx_a1_1_in_v_2 : WORD  // input.input
            input  Application.PLC_PRG.mpx_a1_1_in_v_3 : WORD  // input.input
            input  Application.PLC_PRG.mpx_a1_1_in_freq : WORD  // input.input
            input  Application.PLC_PRG.mpx_a1_1_temp : WORD  // temp.temp
            output Application.PLC_PRG.mpx_a1_test_battery_start : BIT  // battery_test
            output Application.PLC_PRG.mpx_test_battery_command : ARRAY[0..0] OF WORD  // battery_test
            unmapped channels: bypass_out, output, battery, states, input, temp
        MPX_A1_2 : Modbus TCP Slave, 3S - Smart Software Solutions GmbH, version 3.5.4.0
            settings: Unit-ID = 1; ResponseTimeout = 1500; IPAddress = [192, 168, 10, 111]; bypass_out.Function Code = 3; bypass_out.Read Offset = 16#0015; bypass_out.Read Length = 7; bypass_out.Write Offset = 0; bypass_out.Write Length = 0; bypass_out.Cycle Time = 300; output.Function Code = 3; output.Read Offset = 16#001F; output.Read Length = 13; output.Write Offset = 0; output.Write Length = 0; output.Cycle Time = 300; battery.Function Code = 3; battery.Read Offset = 16#002F; battery.Read Length = 7; battery.Write Offset = 0; battery.Write Length = 0; battery.Cycle Time = 300; states.Function Code = 3; states.Read Offset = 16#0000; states.Read Length = 2; states.Write Offset = 0; states.Write Length = 0; states.Cycle Time = 300; input.Function Code = 3; input.Read Offset = 16#000B; input.Read Length = 7; input.Write Offset = 0; input.Write Length = 0; input.Cycle Time = 300; temp.Function Code = 3; temp.Read Offset = 16#003D; temp.Read Length = 1; temp.Write Offset = 0; temp.Write Length = 0; temp.Cycle Time = 300; battery_test.Function Code = 6;
              battery_test.Read Offset = 0; battery_test.Read Length = 0; battery_test.Write Offset = 16#0070; battery_test.Write Length = 1; battery_test.Cycle Time = 100
            input  Application.PLC_PRG.mpx_a1_2_bypass_v_1 : WORD  // bypass_out.bypass_out
            input  Application.PLC_PRG.mpx_a1_2_bypass_v_2 : WORD  // bypass_out.bypass_out
            input  Application.PLC_PRG.mpx_a1_2_bypass_v_3 : WORD  // bypass_out.bypass_out
            input  Application.PLC_PRG.mpx_a1_2_bypass_freq : WORD  // bypass_out.bypass_out
            input  Application.PLC_PRG.mpx_a1_2_output_v_1 : WORD  // bypass_out.bypass_out
            input  Application.PLC_PRG.mpx_a1_2_output_v_2 : WORD  // bypass_out.bypass_out
            input  Application.PLC_PRG.mpx_a1_2_output_v_3 : WORD  // bypass_out.bypass_out
            input  Application.PLC_PRG.mpx_a1_2_output_i_1 : WORD  // output.output
            input  Application.PLC_PRG.mpx_a1_2_output_i_2 : WORD  // output.output
            input  Application.PLC_PRG.mpx_a1_2_output_i_3 : WORD  // output.output
            input  Application.PLC_PRG.mpx_a1_2_load_ph_1 : WORD  // output.output
            input  Application.PLC_PRG.mpx_a1_2_load_ph_2 : WORD  // output.output
            input  Application.PLC_PRG.mpx_a1_2_load_ph_3 : WORD  // output.output
            input  Application.PLC_PRG.mpx_a1_2_output_active_power_1 : WORD  // output.output
            input  Application.PLC_PRG.mpx_a1_2_output_active_power_2 : WORD  // output.output
            input  Application.PLC_PRG.mpx_a1_2_output_active_power_3 : WORD  // output.output
            input  Application.PLC_PRG.mpx_a1_2_output_freq : WORD  // output.output
            input  Application.PLC_PRG.mpx_a1_2_battery_voltage : WORD  // battery.battery
            input  Application.PLC_PRG.mpx_a1_2_battery_current : WORD  // battery.battery
            input  Application.PLC_PRG.mpx_a1_2_battery_capacity : WORD  // battery.battery
            input  Application.PLC_PRG.mpx_a1_2_battery_time : WORD  // battery.battery
            input  Application.PLC_PRG.mpx_a1_2_state_reg_1 : WORD  // states.states
            input  Application.PLC_PRG.mpx_a1_2_state_reg_2 : WORD  // states.states
            input  Application.PLC_PRG.mpx_a1_2_in_v_1 : WORD  // input.input
            input  Application.PLC_PRG.mpx_a1_2_in_v_2 : WORD  // input.input
            input  Application.PLC_PRG.mpx_a1_2_in_v_3 : WORD  // input.input
            input  Application.PLC_PRG.mpx_a1_2_in_freq : WORD  // input.input
            input  Application.PLC_PRG.mpx_a1_2_temp : WORD  // temp.temp
            output Application.PLC_PRG.mpx_a1_test_battery_start : BIT  // battery_test
            output Application.PLC_PRG.mpx_test_battery_command : ARRAY[0..0] OF WORD  // battery_test
            unmapped channels: bypass_out, output, battery, states, input, temp
        MPX_A2_2 : Modbus TCP Slave, 3S - Smart Software Solutions GmbH, version 3.5.4.0
            settings: Unit-ID = 1; ResponseTimeout = 1500; IPAddress = [192, 168, 10, 109]; bypass_out.Function Code = 3; bypass_out.Read Offset = 16#0015; bypass_out.Read Length = 7; bypass_out.Write Offset = 0; bypass_out.Write Length = 0; bypass_out.Cycle Time = 300; output.Function Code = 3; output.Read Offset = 16#001F; output.Read Length = 13; output.Write Offset = 0; output.Write Length = 0; output.Cycle Time = 300; battery.Function Code = 3; battery.Read Offset = 16#002F; battery.Read Length = 7; battery.Write Offset = 0; battery.Write Length = 0; battery.Cycle Time = 300; states.Function Code = 3; states.Read Offset = 16#0000; states.Read Length = 2; states.Write Offset = 0; states.Write Length = 0; states.Cycle Time = 300; input.Function Code = 3; input.Read Offset = 16#000B; input.Read Length = 7; input.Write Offset = 0; input.Write Length = 0; input.Cycle Time = 300; temp.Function Code = 3; temp.Read Offset = 16#003D; temp.Read Length = 1; temp.Write Offset = 0; temp.Write Length = 0; temp.Cycle Time = 300; battery_test.Function Code = 6;
              battery_test.Read Offset = 0; battery_test.Read Length = 0; battery_test.Write Offset = 16#0070; battery_test.Write Length = 1; battery_test.Cycle Time = 100
            input  Application.PLC_PRG.mpx_a2_2_bypass_v_1 : WORD  // bypass_out.bypass_out
            input  Application.PLC_PRG.mpx_a2_2_bypass_v_2 : WORD  // bypass_out.bypass_out
            input  Application.PLC_PRG.mpx_a2_2_bypass_v_3 : WORD  // bypass_out.bypass_out
            input  Application.PLC_PRG.mpx_a2_2_bypass_freq : WORD  // bypass_out.bypass_out
            input  Application.PLC_PRG.mpx_a2_2_output_v_1 : WORD  // bypass_out.bypass_out
            input  Application.PLC_PRG.mpx_a2_2_output_v_2 : WORD  // bypass_out.bypass_out
            input  Application.PLC_PRG.mpx_a2_2_output_v_3 : WORD  // bypass_out.bypass_out
            input  Application.PLC_PRG.mpx_a2_2_output_i_1 : WORD  // output.output
            input  Application.PLC_PRG.mpx_a2_2_output_i_2 : WORD  // output.output
            input  Application.PLC_PRG.mpx_a2_2_output_i_3 : WORD  // output.output
            input  Application.PLC_PRG.mpx_a2_2_load_ph_1 : WORD  // output.output
            input  Application.PLC_PRG.mpx_a2_2_load_ph_2 : WORD  // output.output
            input  Application.PLC_PRG.mpx_a2_2_load_ph_3 : WORD  // output.output
            input  Application.PLC_PRG.mpx_a2_2_output_active_power_1 : WORD  // output.output
            input  Application.PLC_PRG.mpx_a2_2_output_active_power_2 : WORD  // output.output
            input  Application.PLC_PRG.mpx_a2_2_output_active_power_3 : WORD  // output.output
            input  Application.PLC_PRG.mpx_a2_2_output_freq : WORD  // output.output
            input  Application.PLC_PRG.mpx_a2_2_battery_voltage : WORD  // battery.battery
            input  Application.PLC_PRG.mpx_a2_2_battery_current : WORD  // battery.battery
            input  Application.PLC_PRG.mpx_a2_2_battery_capacity : WORD  // battery.battery
            input  Application.PLC_PRG.mpx_a2_2_battery_time : WORD  // battery.battery
            input  Application.PLC_PRG.mpx_a2_2_state_reg_1 : WORD  // states.states
            input  Application.PLC_PRG.mpx_a2_2_state_reg_2 : WORD  // states.states
            input  Application.PLC_PRG.mpx_a2_2_in_v_1 : WORD  // input.input
            input  Application.PLC_PRG.mpx_a2_2_in_v_2 : WORD  // input.input
            input  Application.PLC_PRG.mpx_a2_2_in_v_3 : WORD  // input.input
            input  Application.PLC_PRG.mpx_a2_2_in_freq : WORD  // input.input
            input  Application.PLC_PRG.mpx_a2_2_temp : WORD  // temp.temp
            output Application.PLC_PRG.mpx_a2_test_battery_start : BIT  // battery_test
            output Application.PLC_PRG.mpx_test_battery_command : ARRAY[0..0] OF WORD  // battery_test
            unmapped channels: bypass_out, output, battery, states, input, temp
        MPX_A2_1 : Modbus TCP Slave, 3S - Smart Software Solutions GmbH, version 3.5.4.0
            settings: Unit-ID = 1; ResponseTimeout = 1500; IPAddress = [192, 168, 10, 110]; bypass_out.Function Code = 3; bypass_out.Read Offset = 16#0015; bypass_out.Read Length = 7; bypass_out.Write Offset = 0; bypass_out.Write Length = 0; bypass_out.Cycle Time = 300; output.Function Code = 3; output.Read Offset = 16#001F; output.Read Length = 13; output.Write Offset = 0; output.Write Length = 0; output.Cycle Time = 300; battery.Function Code = 3; battery.Read Offset = 16#002F; battery.Read Length = 7; battery.Write Offset = 0; battery.Write Length = 0; battery.Cycle Time = 300; states.Function Code = 3; states.Read Offset = 16#0000; states.Read Length = 2; states.Write Offset = 0; states.Write Length = 0; states.Cycle Time = 300; input.Function Code = 3; input.Read Offset = 16#000B; input.Read Length = 7; input.Write Offset = 0; input.Write Length = 0; input.Cycle Time = 300; temp.Function Code = 3; temp.Read Offset = 16#003D; temp.Read Length = 1; temp.Write Offset = 0; temp.Write Length = 0; temp.Cycle Time = 300; battery_test.Function Code = 6;
              battery_test.Read Offset = 0; battery_test.Read Length = 0; battery_test.Write Offset = 16#0070; battery_test.Write Length = 1; battery_test.Cycle Time = 100
            input  Application.PLC_PRG.mpx_a2_1_bypass_v_1 : WORD  // bypass_out.bypass_out
            input  Application.PLC_PRG.mpx_a2_1_bypass_v_2 : WORD  // bypass_out.bypass_out
            input  Application.PLC_PRG.mpx_a2_1_bypass_v_3 : WORD  // bypass_out.bypass_out
            input  Application.PLC_PRG.mpx_a2_1_bypass_freq : WORD  // bypass_out.bypass_out
            input  Application.PLC_PRG.mpx_a2_1_output_v_1 : WORD  // bypass_out.bypass_out
            input  Application.PLC_PRG.mpx_a2_1_output_v_2 : WORD  // bypass_out.bypass_out
            input  Application.PLC_PRG.mpx_a2_1_output_v_3 : WORD  // bypass_out.bypass_out
            input  Application.PLC_PRG.mpx_a2_1_output_i_1 : WORD  // output.output
            input  Application.PLC_PRG.mpx_a2_1_output_i_2 : WORD  // output.output
            input  Application.PLC_PRG.mpx_a2_1_output_i_3 : WORD  // output.output
            input  Application.PLC_PRG.mpx_a2_1_load_ph_1 : WORD  // output.output
            input  Application.PLC_PRG.mpx_a2_1_load_ph_2 : WORD  // output.output
            input  Application.PLC_PRG.mpx_a2_1_load_ph_3 : WORD  // output.output
            input  Application.PLC_PRG.mpx_a2_1_output_active_power_1 : WORD  // output.output
            input  Application.PLC_PRG.mpx_a2_1_output_active_power_2 : WORD  // output.output
            input  Application.PLC_PRG.mpx_a2_1_output_active_power_3 : WORD  // output.output
            input  Application.PLC_PRG.mpx_a2_1_output_freq : WORD  // output.output
            input  Application.PLC_PRG.mpx_a2_1_battery_voltage : WORD  // battery.battery
            input  Application.PLC_PRG.mpx_a2_1_battery_current : WORD  // battery.battery
            input  Application.PLC_PRG.mpx_a2_1_battery_capacity : WORD  // battery.battery
            input  Application.PLC_PRG.mpx_a2_1_battery_time : WORD  // battery.battery
            input  Application.PLC_PRG.mpx_a2_1_state_reg_1 : WORD  // states.states
            input  Application.PLC_PRG.mpx_a2_1_state_reg_2 : WORD  // states.states
            input  Application.PLC_PRG.mpx_a2_1_in_v_1 : WORD  // input.input
            input  Application.PLC_PRG.mpx_a2_1_in_v_2 : WORD  // input.input
            input  Application.PLC_PRG.mpx_a2_1_in_v_3 : WORD  // input.input
            input  Application.PLC_PRG.mpx_a2_1_in_freq : WORD  // input.input
            input  Application.PLC_PRG.mpx_a2_1_temp : WORD  // temp.temp
            output Application.PLC_PRG.mpx_a2_test_battery_start : BIT  // battery_test
            output Application.PLC_PRG.mpx_test_battery_command : ARRAY[0..0] OF WORD  // battery_test
            unmapped channels: bypass_out, output, battery, states, input, temp
    ModbusIN : Modbus COM, 3S - Smart Software Solutions GmbH, version 3.4.0.0
        settings: DataBits = 8; StopBits = 1; ComPort = 1
      ModbusMaster : Modbus Master, COM Port, 3S - Smart Software Solutions GmbH, version 3.5.5.0
          settings: Transmission = 'RTU'; ResponseTimeout = 1000; TimeBetweenFrames = 50; Auto-restart communication = TRUE
        MV_110 : Modbus Slave, COM Port, 3S - Smart Software Solutions GmbH, version 3.5.4.0
            settings: SlaveAddress = 2; ResponseTimeout = 1000; UseExtendedFunctionCodes = TRUE; Channel 0.Function Code = 3; Channel 0.Read Offset = 16#0033; Channel 0.Read Length = 1; Channel 0.Write Offset = 0; Channel 0.Write Length = 0; Channel 0.Cycle Time = 500
            input  Application.PLC_PRG.mv110_reg : ARRAY[0..0] OF WORD  // Channel 0
        PLC : Modbus Slave, COM Port, 3S - Smart Software Solutions GmbH, version 3.5.4.0
            settings: SlaveAddress = 1; ResponseTimeout = 1000; UseExtendedFunctionCodes = TRUE; Channel 0.Function Code = 3; Channel 0.Read Offset = 16#0000; Channel 0.Read Length = 3; Channel 0.Write Offset = 0; Channel 0.Write Length = 0; Channel 0.Cycle Time = 500
            input  Application.PLC_PRG.climate_temp_in : WORD  // Channel 0.Channel 0
            input  Application.PLC_PRG.climate_temp_out : WORD  // Channel 0.Channel 0
            input  Application.PLC_PRG.climate_state_reg : WORD  // Channel 0.Channel 0
            unmapped channels: Channel 0
    ModbusOUT : Modbus COM, 3S - Smart Software Solutions GmbH, version 3.4.0.0
        settings: DataBits = 8; StopBits = 1; ComPort = 2
      Modbus_Serial_Device : Modbus Serial Device, 3S - Smart Software Solutions GmbH, version 3.5.5.0
          output Application.PLC_PRG.mpx_s1_1_battery_capacity : WORD  // Outputs.Outputs
          output Application.PLC_PRG.mpx_s1_1_battery_current : WORD  // Outputs.Outputs
          output Application.PLC_PRG.mpx_s1_1_battery_time : WORD  // Outputs.Outputs
          output Application.PLC_PRG.mpx_s1_1_battery_voltage : WORD  // Outputs.Outputs
          output Application.PLC_PRG.mpx_s1_1_bypass_freq : WORD  // Outputs.Outputs
          output Application.PLC_PRG.mpx_s1_1_bypass_v_1 : WORD  // Outputs.Outputs
          output Application.PLC_PRG.mpx_s1_1_bypass_v_2 : WORD  // Outputs.Outputs
          output Application.PLC_PRG.mpx_s1_1_bypass_v_3 : WORD  // Outputs.Outputs
          output Application.PLC_PRG.mpx_s1_1_in_freq : WORD  // Outputs.Outputs
          output Application.PLC_PRG.mpx_s1_1_in_v_1 : WORD  // Outputs.Outputs
          output Application.PLC_PRG.mpx_s1_1_in_v_2 : WORD  // Outputs.Outputs
          output Application.PLC_PRG.mpx_s1_1_in_v_3 : WORD  // Outputs.Outputs
          output Application.PLC_PRG.mpx_s1_1_load_ph_1 : WORD  // Outputs.Outputs
          output Application.PLC_PRG.mpx_s1_1_load_ph_2 : WORD  // Outputs.Outputs
          output Application.PLC_PRG.mpx_s1_1_load_ph_3 : WORD  // Outputs.Outputs
          output Application.PLC_PRG.mpx_s1_1_output_active_power_1 : WORD  // Outputs.Outputs
          output Application.PLC_PRG.mpx_s1_1_output_active_power_2 : WORD  // Outputs.Outputs
          output Application.PLC_PRG.mpx_s1_1_output_active_power_3 : WORD  // Outputs.Outputs
          output Application.PLC_PRG.mpx_s1_1_output_freq : WORD  // Outputs.Outputs
          output Application.PLC_PRG.mpx_s1_1_output_i_1 : WORD  // Outputs.Outputs
          output Application.PLC_PRG.mpx_s1_1_output_i_2 : WORD  // Outputs.Outputs
          output Application.PLC_PRG.mpx_s1_1_output_i_3 : WORD  // Outputs.Outputs
          output Application.PLC_PRG.mpx_s1_1_output_v_1 : WORD  // Outputs.Outputs
          output Application.PLC_PRG.mpx_s1_1_output_v_2 : WORD  // Outputs.Outputs
          output Application.PLC_PRG.mpx_s1_1_output_v_3 : WORD  // Outputs.Outputs
          output Application.PLC_PRG.mpx_s1_1_state_reg_1 : WORD  // Outputs.Outputs
          output Application.PLC_PRG.mpx_s1_1_state_reg_2 : WORD  // Outputs.Outputs
          output Application.PLC_PRG.mpx_s1_1_temp : WORD  // Outputs.Outputs
          output Application.PLC_PRG.mpx_s1_2_battery_capacity : WORD  // Outputs.Outputs
          output Application.PLC_PRG.mpx_s1_2_battery_current : WORD  // Outputs.Outputs
          output Application.PLC_PRG.mpx_s1_2_battery_time : WORD  // Outputs.Outputs
          output Application.PLC_PRG.mpx_s1_2_battery_voltage : WORD  // Outputs.Outputs
          output Application.PLC_PRG.mpx_s1_2_bypass_freq : WORD  // Outputs.Outputs
          output Application.PLC_PRG.mpx_s1_2_bypass_v_1 : WORD  // Outputs.Outputs
          output Application.PLC_PRG.mpx_s1_2_bypass_v_2 : WORD  // Outputs.Outputs
          output Application.PLC_PRG.mpx_s1_2_bypass_v_3 : WORD  // Outputs.Outputs
          output Application.PLC_PRG.mpx_s1_2_in_freq : WORD  // Outputs.Outputs
          output Application.PLC_PRG.mpx_s1_2_in_v_1 : WORD  // Outputs.Outputs
          output Application.PLC_PRG.mpx_s1_2_in_v_2 : WORD  // Outputs.Outputs
          output Application.PLC_PRG.mpx_s1_2_in_v_3 : WORD  // Outputs.Outputs
          output Application.PLC_PRG.mpx_s1_2_load_ph_1 : WORD  // Outputs.Outputs
          output Application.PLC_PRG.mpx_s1_2_load_ph_2 : WORD  // Outputs.Outputs
          output Application.PLC_PRG.mpx_s1_2_load_ph_3 : WORD  // Outputs.Outputs
          output Application.PLC_PRG.mpx_s1_2_output_active_power_1 : WORD  // Outputs.Outputs
          output Application.PLC_PRG.mpx_s1_2_output_active_power_2 : WORD  // Outputs.Outputs
          output Application.PLC_PRG.mpx_s1_2_output_active_power_3 : WORD  // Outputs.Outputs
          output Application.PLC_PRG.mpx_s1_2_output_freq : WORD  // Outputs.Outputs
          output Application.PLC_PRG.mpx_s1_2_output_i_1 : WORD  // Outputs.Outputs
          output Application.PLC_PRG.mpx_s1_2_output_i_2 : WORD  // Outputs.Outputs
          output Application.PLC_PRG.mpx_s1_2_output_i_3 : WORD  // Outputs.Outputs
          output Application.PLC_PRG.mpx_s1_2_output_v_1 : WORD  // Outputs.Outputs
          output Application.PLC_PRG.mpx_s1_2_output_v_2 : WORD  // Outputs.Outputs
          output Application.PLC_PRG.mpx_s1_2_output_v_3 : WORD  // Outputs.Outputs
          output Application.PLC_PRG.mpx_s1_2_state_reg_1 : WORD  // Outputs.Outputs
          output Application.PLC_PRG.mpx_s1_2_state_reg_2 : WORD  // Outputs.Outputs
          output Application.PLC_PRG.mpx_s1_2_temp : WORD  // Outputs.Outputs
          output Application.PLC_PRG.mpx_s1_3_battery_capacity : WORD  // Outputs.Outputs
          output Application.PLC_PRG.mpx_s1_3_battery_current : WORD  // Outputs.Outputs
          output Application.PLC_PRG.mpx_s1_3_battery_time : WORD  // Outputs.Outputs
          output Application.PLC_PRG.mpx_s1_3_battery_voltage : WORD  // Outputs.Outputs
          output Application.PLC_PRG.mpx_s1_3_bypass_freq : WORD  // Outputs.Outputs
          output Application.PLC_PRG.mpx_s1_3_bypass_v_1 : WORD  // Outputs.Outputs
          output Application.PLC_PRG.mpx_s1_3_bypass_v_2 : WORD  // Outputs.Outputs
          output Application.PLC_PRG.mpx_s1_3_bypass_v_3 : WORD  // Outputs.Outputs
          output Application.PLC_PRG.mpx_s1_3_in_freq : WORD  // Outputs.Outputs
          output Application.PLC_PRG.mpx_s1_3_in_v_1 : WORD  // Outputs.Outputs
          output Application.PLC_PRG.mpx_s1_3_in_v_2 : WORD  // Outputs.Outputs
          output Application.PLC_PRG.mpx_s1_3_in_v_3 : WORD  // Outputs.Outputs
          output Application.PLC_PRG.mpx_s1_3_load_ph_1 : WORD  // Outputs.Outputs
          output Application.PLC_PRG.mpx_s1_3_load_ph_2 : WORD  // Outputs.Outputs
          output Application.PLC_PRG.mpx_s1_3_load_ph_3 : WORD  // Outputs.Outputs
          output Application.PLC_PRG.mpx_s1_3_output_active_power_1 : WORD  // Outputs.Outputs
          output Application.PLC_PRG.mpx_s1_3_output_active_power_2 : WORD  // Outputs.Outputs
          output Application.PLC_PRG.mpx_s1_3_output_active_power_3 : WORD  // Outputs.Outputs
          output Application.PLC_PRG.mpx_s1_3_output_freq : WORD  // Outputs.Outputs
          output Application.PLC_PRG.mpx_s1_3_output_i_1 : WORD  // Outputs.Outputs
          output Application.PLC_PRG.mpx_s1_3_output_i_2 : WORD  // Outputs.Outputs
          output Application.PLC_PRG.mpx_s1_3_output_i_3 : WORD  // Outputs.Outputs
          output Application.PLC_PRG.mpx_s1_3_output_v_1 : WORD  // Outputs.Outputs
          output Application.PLC_PRG.mpx_s1_3_output_v_2 : WORD  // Outputs.Outputs
          output Application.PLC_PRG.mpx_s1_3_output_v_3 : WORD  // Outputs.Outputs
          output Application.PLC_PRG.mpx_s1_3_state_reg_1 : WORD  // Outputs.Outputs
          output Application.PLC_PRG.mpx_s1_3_state_reg_2 : WORD  // Outputs.Outputs
          output Application.PLC_PRG.mpx_s1_3_temp : WORD  // Outputs.Outputs
          output Application.PLC_PRG.mpx_s1_4_battery_capacity : WORD  // Outputs.Outputs
          output Application.PLC_PRG.mpx_s1_4_battery_current : WORD  // Outputs.Outputs
          output Application.PLC_PRG.mpx_s1_4_battery_time : WORD  // Outputs.Outputs
          output Application.PLC_PRG.mpx_s1_4_battery_voltage : WORD  // Outputs.Outputs
          output Application.PLC_PRG.mpx_s1_4_bypass_freq : WORD  // Outputs.Outputs
          output Application.PLC_PRG.mpx_s1_4_bypass_v_1 : WORD  // Outputs.Outputs
          output Application.PLC_PRG.mpx_s1_4_bypass_v_2 : WORD  // Outputs.Outputs
          output Application.PLC_PRG.mpx_s1_4_bypass_v_3 : WORD  // Outputs.Outputs
          output Application.PLC_PRG.mpx_s1_4_in_freq : WORD  // Outputs.Outputs
          output Application.PLC_PRG.mpx_s1_4_in_v_1 : WORD  // Outputs.Outputs
          output Application.PLC_PRG.mpx_s1_4_in_v_2 : WORD  // Outputs.Outputs
          output Application.PLC_PRG.mpx_s1_4_in_v_3 : WORD  // Outputs.Outputs
          output Application.PLC_PRG.mpx_s1_4_load_ph_1 : WORD  // Outputs.Outputs
          output Application.PLC_PRG.mpx_s1_4_load_ph_2 : WORD  // Outputs.Outputs
          output Application.PLC_PRG.mpx_s1_4_load_ph_3 : WORD  // Outputs.Outputs
          output Application.PLC_PRG.mpx_s1_4_output_active_power_1 : WORD  // Outputs.Outputs
          output Application.PLC_PRG.mpx_s1_4_output_active_power_2 : WORD  // Outputs.Outputs
          output Application.PLC_PRG.mpx_s1_4_output_active_power_3 : WORD  // Outputs.Outputs
          output Application.PLC_PRG.mpx_s1_4_output_freq : WORD  // Outputs.Outputs
          output Application.PLC_PRG.mpx_s1_4_output_i_1 : WORD  // Outputs.Outputs
          output Application.PLC_PRG.mpx_s1_4_output_i_2 : WORD  // Outputs.Outputs
          output Application.PLC_PRG.mpx_s1_4_output_i_3 : WORD  // Outputs.Outputs
          output Application.PLC_PRG.mpx_s1_4_output_v_1 : WORD  // Outputs.Outputs
          output Application.PLC_PRG.mpx_s1_4_output_v_2 : WORD  // Outputs.Outputs
          output Application.PLC_PRG.mpx_s1_4_output_v_3 : WORD  // Outputs.Outputs
          output Application.PLC_PRG.mpx_s1_4_state_reg_1 : WORD  // Outputs.Outputs
          output Application.PLC_PRG.mpx_s1_4_state_reg_2 : WORD  // Outputs.Outputs
          output Application.PLC_PRG.mpx_s1_4_temp : WORD  // Outputs.Outputs
          output Application.PLC_PRG.mpx_s2_1_battery_capacity : WORD  // Outputs.Outputs
          output Application.PLC_PRG.mpx_s2_1_battery_current : WORD  // Outputs.Outputs
          output Application.PLC_PRG.mpx_s2_1_battery_time : WORD  // Outputs.Outputs
          output Application.PLC_PRG.mpx_s2_1_battery_voltage : WORD  // Outputs.Outputs
          output Application.PLC_PRG.mpx_s2_1_bypass_freq : WORD  // Outputs.Outputs
          output Application.PLC_PRG.mpx_s2_1_bypass_v_1 : WORD  // Outputs.Outputs
          output Application.PLC_PRG.mpx_s2_1_bypass_v_2 : WORD  // Outputs.Outputs
          output Application.PLC_PRG.mpx_s2_1_bypass_v_3 : WORD  // Outputs.Outputs
          output Application.PLC_PRG.mpx_s2_1_in_freq : WORD  // Outputs.Outputs
          output Application.PLC_PRG.mpx_s2_1_in_v_1 : WORD  // Outputs.Outputs
          output Application.PLC_PRG.mpx_s2_1_in_v_2 : WORD  // Outputs.Outputs
          output Application.PLC_PRG.mpx_s2_1_in_v_3 : WORD  // Outputs.Outputs
          output Application.PLC_PRG.mpx_s2_1_load_ph_1 : WORD  // Outputs.Outputs
          output Application.PLC_PRG.mpx_s2_1_load_ph_2 : WORD  // Outputs.Outputs
          output Application.PLC_PRG.mpx_s2_1_load_ph_3 : WORD  // Outputs.Outputs
          output Application.PLC_PRG.mpx_s2_1_output_active_power_1 : WORD  // Outputs.Outputs
          output Application.PLC_PRG.mpx_s2_1_output_active_power_2 : WORD  // Outputs.Outputs
          output Application.PLC_PRG.mpx_s2_1_output_active_power_3 : WORD  // Outputs.Outputs
          output Application.PLC_PRG.mpx_s2_1_output_freq : WORD  // Outputs.Outputs
          output Application.PLC_PRG.mpx_s2_1_output_i_1 : WORD  // Outputs.Outputs
          output Application.PLC_PRG.mpx_s2_1_output_i_2 : WORD  // Outputs.Outputs
          output Application.PLC_PRG.mpx_s2_1_output_i_3 : WORD  // Outputs.Outputs
          output Application.PLC_PRG.mpx_s2_1_output_v_1 : WORD  // Outputs.Outputs
          output Application.PLC_PRG.mpx_s2_1_output_v_2 : WORD  // Outputs.Outputs
          output Application.PLC_PRG.mpx_s2_1_output_v_3 : WORD  // Outputs.Outputs
          output Application.PLC_PRG.mpx_s2_1_state_reg_1 : WORD  // Outputs.Outputs
          output Application.PLC_PRG.mpx_s2_1_state_reg_2 : WORD  // Outputs.Outputs
          output Application.PLC_PRG.mpx_s2_1_temp : WORD  // Outputs.Outputs
          output Application.PLC_PRG.mpx_s2_2_battery_capacity : WORD  // Outputs.Outputs
          output Application.PLC_PRG.mpx_s2_2_battery_current : WORD  // Outputs.Outputs
          output Application.PLC_PRG.mpx_s2_2_battery_time : WORD  // Outputs.Outputs
          output Application.PLC_PRG.mpx_s2_2_battery_voltage : WORD  // Outputs.Outputs
          output Application.PLC_PRG.mpx_s2_2_bypass_freq : WORD  // Outputs.Outputs
          output Application.PLC_PRG.mpx_s2_2_bypass_v_1 : WORD  // Outputs.Outputs
          output Application.PLC_PRG.mpx_s2_2_bypass_v_2 : WORD  // Outputs.Outputs
          output Application.PLC_PRG.mpx_s2_2_bypass_v_3 : WORD  // Outputs.Outputs
          output Application.PLC_PRG.mpx_s2_2_in_freq : WORD  // Outputs.Outputs
          output Application.PLC_PRG.mpx_s2_2_in_v_1 : WORD  // Outputs.Outputs
          output Application.PLC_PRG.mpx_s2_2_in_v_2 : WORD  // Outputs.Outputs
          output Application.PLC_PRG.mpx_s2_2_in_v_3 : WORD  // Outputs.Outputs
          output Application.PLC_PRG.mpx_s2_2_load_ph_1 : WORD  // Outputs.Outputs
          output Application.PLC_PRG.mpx_s2_2_load_ph_2 : WORD  // Outputs.Outputs
          output Application.PLC_PRG.mpx_s2_2_load_ph_3 : WORD  // Outputs.Outputs
          output Application.PLC_PRG.mpx_s2_2_output_active_power_1 : WORD  // Outputs.Outputs
          output Application.PLC_PRG.mpx_s2_2_output_active_power_2 : WORD  // Outputs.Outputs
          output Application.PLC_PRG.mpx_s2_2_output_active_power_3 : WORD  // Outputs.Outputs
          output Application.PLC_PRG.mpx_s2_2_output_freq : WORD  // Outputs.Outputs
          output Application.PLC_PRG.mpx_s2_2_output_i_1 : WORD  // Outputs.Outputs
          output Application.PLC_PRG.mpx_s2_2_output_i_2 : WORD  // Outputs.Outputs
          output Application.PLC_PRG.mpx_s2_2_output_i_3 : WORD  // Outputs.Outputs
          output Application.PLC_PRG.mpx_s2_2_output_v_1 : WORD  // Outputs.Outputs
          output Application.PLC_PRG.mpx_s2_2_output_v_2 : WORD  // Outputs.Outputs
          output Application.PLC_PRG.mpx_s2_2_output_v_3 : WORD  // Outputs.Outputs
          output Application.PLC_PRG.mpx_s2_2_state_reg_1 : WORD  // Outputs.Outputs
          output Application.PLC_PRG.mpx_s2_2_state_reg_2 : WORD  // Outputs.Outputs
          output Application.PLC_PRG.mpx_s2_2_temp : WORD  // Outputs.Outputs
          output Application.PLC_PRG.mpx_s2_3_battery_capacity : WORD  // Outputs.Outputs
          output Application.PLC_PRG.mpx_s2_3_battery_current : WORD  // Outputs.Outputs
          output Application.PLC_PRG.mpx_s2_3_battery_time : WORD  // Outputs.Outputs
          output Application.PLC_PRG.mpx_s2_3_battery_voltage : WORD  // Outputs.Outputs
          output Application.PLC_PRG.mpx_s2_3_bypass_freq : WORD  // Outputs.Outputs
          output Application.PLC_PRG.mpx_s2_3_bypass_v_1 : WORD  // Outputs.Outputs
          output Application.PLC_PRG.mpx_s2_3_bypass_v_2 : WORD  // Outputs.Outputs
          output Application.PLC_PRG.mpx_s2_3_bypass_v_3 : WORD  // Outputs.Outputs
          output Application.PLC_PRG.mpx_s2_3_in_freq : WORD  // Outputs.Outputs
          output Application.PLC_PRG.mpx_s2_3_in_v_1 : WORD  // Outputs.Outputs
          output Application.PLC_PRG.mpx_s2_3_in_v_2 : WORD  // Outputs.Outputs
          output Application.PLC_PRG.mpx_s2_3_in_v_3 : WORD  // Outputs.Outputs
          output Application.PLC_PRG.mpx_s2_3_load_ph_1 : WORD  // Outputs.Outputs
          output Application.PLC_PRG.mpx_s2_3_load_ph_2 : WORD  // Outputs.Outputs
          output Application.PLC_PRG.mpx_s2_3_load_ph_3 : WORD  // Outputs.Outputs
          output Application.PLC_PRG.mpx_s2_3_output_active_power_1 : WORD  // Outputs.Outputs
          output Application.PLC_PRG.mpx_s2_3_output_active_power_2 : WORD  // Outputs.Outputs
          output Application.PLC_PRG.mpx_s2_3_output_active_power_3 : WORD  // Outputs.Outputs
          output Application.PLC_PRG.mpx_s2_3_output_freq : WORD  // Outputs.Outputs
          output Application.PLC_PRG.mpx_s2_3_output_i_1 : WORD  // Outputs.Outputs
          output Application.PLC_PRG.mpx_s2_3_output_i_2 : WORD  // Outputs.Outputs
          output Application.PLC_PRG.mpx_s2_3_output_i_3 : WORD  // Outputs.Outputs
          output Application.PLC_PRG.mpx_s2_3_output_v_1 : WORD  // Outputs.Outputs
          output Application.PLC_PRG.mpx_s2_3_output_v_2 : WORD  // Outputs.Outputs
          output Application.PLC_PRG.mpx_s2_3_output_v_3 : WORD  // Outputs.Outputs
          output Application.PLC_PRG.mpx_s2_3_state_reg_1 : WORD  // Outputs.Outputs
          output Application.PLC_PRG.mpx_s2_3_state_reg_2 : WORD  // Outputs.Outputs
          output Application.PLC_PRG.mpx_s2_3_temp : WORD  // Outputs.Outputs
          output Application.PLC_PRG.mpx_s2_4_battery_capacity : WORD  // Outputs.Outputs
          output Application.PLC_PRG.mpx_s2_4_battery_current : WORD  // Outputs.Outputs
          output Application.PLC_PRG.mpx_s2_4_battery_time : WORD  // Outputs.Outputs
          output Application.PLC_PRG.mpx_s2_4_battery_voltage : WORD  // Outputs.Outputs
          output Application.PLC_PRG.mpx_s2_4_bypass_freq : WORD  // Outputs.Outputs
          output Application.PLC_PRG.mpx_s2_4_bypass_v_1 : WORD  // Outputs.Outputs
          output Application.PLC_PRG.mpx_s2_4_bypass_v_2 : WORD  // Outputs.Outputs
          output Application.PLC_PRG.mpx_s2_4_bypass_v_3 : WORD  // Outputs.Outputs
          output Application.PLC_PRG.mpx_s2_4_in_freq : WORD  // Outputs.Outputs
          output Application.PLC_PRG.mpx_s2_4_in_v_1 : WORD  // Outputs.Outputs
          output Application.PLC_PRG.mpx_s2_4_in_v_2 : WORD  // Outputs.Outputs
          output Application.PLC_PRG.mpx_s2_4_in_v_3 : WORD  // Outputs.Outputs
          output Application.PLC_PRG.mpx_s2_4_load_ph_1 : WORD  // Outputs.Outputs
          output Application.PLC_PRG.mpx_s2_4_load_ph_2 : WORD  // Outputs.Outputs
          output Application.PLC_PRG.mpx_s2_4_load_ph_3 : WORD  // Outputs.Outputs
          output Application.PLC_PRG.mpx_s2_4_output_active_power_1 : WORD  // Outputs.Outputs
          output Application.PLC_PRG.mpx_s2_4_output_active_power_2 : WORD  // Outputs.Outputs
          output Application.PLC_PRG.mpx_s2_4_output_active_power_3 : WORD  // Outputs.Outputs
          output Application.PLC_PRG.mpx_s2_4_output_freq : WORD  // Outputs.Outputs
          output Application.PLC_PRG.mpx_s2_4_output_i_1 : WORD  // Outputs.Outputs
          output Application.PLC_PRG.mpx_s2_4_output_i_2 : WORD  // Outputs.Outputs
          output Application.PLC_PRG.mpx_s2_4_output_i_3 : WORD  // Outputs.Outputs
          output Application.PLC_PRG.mpx_s2_4_output_v_1 : WORD  // Outputs.Outputs
          output Application.PLC_PRG.mpx_s2_4_output_v_2 : WORD  // Outputs.Outputs
          output Application.PLC_PRG.mpx_s2_4_output_v_3 : WORD  // Outputs.Outputs
          output Application.PLC_PRG.mpx_s2_4_state_reg_1 : WORD  // Outputs.Outputs
          output Application.PLC_PRG.mpx_s2_4_state_reg_2 : WORD  // Outputs.Outputs
          output Application.PLC_PRG.mpx_s2_4_temp : WORD  // Outputs.Outputs
          output Application.PLC_PRG.mpx_a1_1_battery_capacity : WORD  // Outputs.Outputs
          output Application.PLC_PRG.mpx_a1_1_battery_current : WORD  // Outputs.Outputs
          output Application.PLC_PRG.mpx_a1_1_battery_time : WORD  // Outputs.Outputs
          output Application.PLC_PRG.mpx_a1_1_battery_voltage : WORD  // Outputs.Outputs
          output Application.PLC_PRG.mpx_a1_1_bypass_freq : WORD  // Outputs.Outputs
          output Application.PLC_PRG.mpx_a1_1_bypass_v_1 : WORD  // Outputs.Outputs
          output Application.PLC_PRG.mpx_a1_1_in_freq : WORD  // Outputs.Outputs
          output Application.PLC_PRG.mpx_a1_1_in_v_1 : WORD  // Outputs.Outputs
          output Application.PLC_PRG.mpx_a1_1_in_v_2 : WORD  // Outputs.Outputs
          output Application.PLC_PRG.mpx_a1_1_in_v_3 : WORD  // Outputs.Outputs
          output Application.PLC_PRG.mpx_a1_1_load_ph_1 : WORD  // Outputs.Outputs
          output Application.PLC_PRG.mpx_a1_1_output_active_power_1 : WORD  // Outputs.Outputs
          output Application.PLC_PRG.mpx_a1_1_output_freq : WORD  // Outputs.Outputs
          output Application.PLC_PRG.mpx_a1_1_output_i_1 : WORD  // Outputs.Outputs
          output Application.PLC_PRG.mpx_a1_1_output_v_1 : WORD  // Outputs.Outputs
          output Application.PLC_PRG.mpx_a1_1_state_reg_1 : WORD  // Outputs.Outputs
          output Application.PLC_PRG.mpx_a1_1_state_reg_2 : WORD  // Outputs.Outputs
          output Application.PLC_PRG.mpx_a1_1_temp : WORD  // Outputs.Outputs
          output Application.PLC_PRG.mpx_a1_2_battery_capacity : WORD  // Outputs.Outputs
          output Application.PLC_PRG.mpx_a1_2_battery_current : WORD  // Outputs.Outputs
          output Application.PLC_PRG.mpx_a1_2_battery_time : WORD  // Outputs.Outputs
          output Application.PLC_PRG.mpx_a1_2_battery_voltage : WORD  // Outputs.Outputs
          output Application.PLC_PRG.mpx_a1_2_bypass_freq : WORD  // Outputs.Outputs
          output Application.PLC_PRG.mpx_a1_2_bypass_v_1 : WORD  // Outputs.Outputs
          output Application.PLC_PRG.mpx_a1_2_in_freq : WORD  // Outputs.Outputs
          output Application.PLC_PRG.mpx_a1_2_in_v_1 : WORD  // Outputs.Outputs
          output Application.PLC_PRG.mpx_a1_2_in_v_2 : WORD  // Outputs.Outputs
          output Application.PLC_PRG.mpx_a1_2_in_v_3 : WORD  // Outputs.Outputs
          output Application.PLC_PRG.mpx_a1_2_load_ph_1 : WORD  // Outputs.Outputs
          output Application.PLC_PRG.mpx_a1_2_output_active_power_1 : WORD  // Outputs.Outputs
          output Application.PLC_PRG.mpx_a1_2_output_freq : WORD  // Outputs.Outputs
          output Application.PLC_PRG.mpx_a1_2_output_i_1 : WORD  // Outputs.Outputs
          output Application.PLC_PRG.mpx_a1_2_output_v_1 : WORD  // Outputs.Outputs
          output Application.PLC_PRG.mpx_a1_2_state_reg_1 : WORD  // Outputs.Outputs
          output Application.PLC_PRG.mpx_a1_2_state_reg_2 : WORD  // Outputs.Outputs
          output Application.PLC_PRG.mpx_a1_2_temp : WORD  // Outputs.Outputs
          output Application.PLC_PRG.mpx_a2_1_battery_capacity : WORD  // Outputs.Outputs
          output Application.PLC_PRG.mpx_a2_1_battery_current : WORD  // Outputs.Outputs
          output Application.PLC_PRG.mpx_a2_1_battery_time : WORD  // Outputs.Outputs
          output Application.PLC_PRG.mpx_a2_1_battery_voltage : WORD  // Outputs.Outputs
          output Application.PLC_PRG.mpx_a2_1_bypass_freq : WORD  // Outputs.Outputs
          output Application.PLC_PRG.mpx_a2_1_bypass_v_1 : WORD  // Outputs.Outputs
          output Application.PLC_PRG.mpx_a2_1_in_freq : WORD  // Outputs.Outputs
          output Application.PLC_PRG.mpx_a2_1_in_v_1 : WORD  // Outputs.Outputs
          output Application.PLC_PRG.mpx_a2_1_in_v_2 : WORD  // Outputs.Outputs
          output Application.PLC_PRG.mpx_a2_1_in_v_3 : WORD  // Outputs.Outputs
          output Application.PLC_PRG.mpx_a2_1_load_ph_1 : WORD  // Outputs.Outputs
          output Application.PLC_PRG.mpx_a2_1_output_active_power_1 : WORD  // Outputs.Outputs
          output Application.PLC_PRG.mpx_a2_1_output_freq : WORD  // Outputs.Outputs
          output Application.PLC_PRG.mpx_a2_1_output_i_1 : WORD  // Outputs.Outputs
          output Application.PLC_PRG.mpx_a2_1_output_v_1 : WORD  // Outputs.Outputs
          output Application.PLC_PRG.mpx_a2_1_state_reg_1 : WORD  // Outputs.Outputs
          output Application.PLC_PRG.mpx_a2_1_state_reg_2 : WORD  // Outputs.Outputs
          output Application.PLC_PRG.mpx_a2_1_temp : WORD  // Outputs.Outputs
          output Application.PLC_PRG.mpx_a2_2_battery_capacity : WORD  // Outputs.Outputs
          output Application.PLC_PRG.mpx_a2_2_battery_current : WORD  // Outputs.Outputs
          output Application.PLC_PRG.mpx_a2_2_battery_time : WORD  // Outputs.Outputs
          output Application.PLC_PRG.mpx_a2_2_battery_voltage : WORD  // Outputs.Outputs
          output Application.PLC_PRG.mpx_a2_2_bypass_freq : WORD  // Outputs.Outputs
          output Application.PLC_PRG.mpx_a2_2_bypass_v_1 : WORD  // Outputs.Outputs
          output Application.PLC_PRG.mpx_a2_2_in_freq : WORD  // Outputs.Outputs
          output Application.PLC_PRG.mpx_a2_2_in_v_1 : WORD  // Outputs.Outputs
          output Application.PLC_PRG.mpx_a2_2_in_v_2 : WORD  // Outputs.Outputs
          output Application.PLC_PRG.mpx_a2_2_in_v_3 : WORD  // Outputs.Outputs
          output Application.PLC_PRG.mpx_a2_2_load_ph_1 : WORD  // Outputs.Outputs
          output Application.PLC_PRG.mpx_a2_2_output_active_power_1 : WORD  // Outputs.Outputs
          output Application.PLC_PRG.mpx_a2_2_output_freq : WORD  // Outputs.Outputs
          output Application.PLC_PRG.mpx_a2_2_output_i_1 : WORD  // Outputs.Outputs
          output Application.PLC_PRG.mpx_a2_2_output_v_1 : WORD  // Outputs.Outputs
          output Application.PLC_PRG.mpx_a2_2_state_reg_1 : WORD  // Outputs.Outputs
          output Application.PLC_PRG.mpx_a2_2_state_reg_2 : WORD  // Outputs.Outputs
          output Application.PLC_PRG.mpx_a2_2_temp : WORD  // Outputs.Outputs
          output Application.GPIO_HANDLER.IN_1 : BOOL  // Outputs.Outputs.Bit0
          output Application.GPIO_HANDLER.IN_2 : BOOL  // Outputs.Outputs.Bit1
          output Application.GPIO_HANDLER.IN_3 : BOOL  // Outputs.Outputs.Bit2
          output Application.PLC_PRG.climate_temp_excess : BOOL  // Outputs.Outputs.Bit3
          output Application.PLC_PRG.mv110_in_0_in_main_present : BOOL  // Outputs.Outputs.Bit4
          output Application.PLC_PRG.mv110_in_1_in_reserve_present : BOOL  // Outputs.Outputs.Bit5
          output Application.PLC_PRG.mv110_in_2_bp_sn_present : BOOL  // Outputs.Outputs.Bit6
          output Application.PLC_PRG.mv110_in_3_gp_sn_present : BOOL  // Outputs.Outputs.Bit7
          output Application.PLC_PRG.mv110_in_4_qs1_1position : BOOL  // Outputs.Outputs.Bit8
          output Application.PLC_PRG.mv110_in_5_qs1_2position : BOOL  // Outputs.Outputs.Bit9
          output Application.PLC_PRG.mv110_in_7_gp1_u_fault : BOOL  // Outputs.Outputs.Bit10
          output Application.PLC_PRG.mv110_in_8_gp2_u_fault : BOOL  // Outputs.Outputs.Bit11
          output Application.GPIO_HANDLER.IN_4 : BOOL  // Outputs.Outputs.Bit12
          output Application.GPIO_HANDLER.IN_5 : BOOL  // Outputs.Outputs.Bit13
          output Application.GPIO_HANDLER.IN_6 : BOOL  // Outputs.Outputs.Bit14
          output Application.GPIO_HANDLER.IN_7 : BOOL  // Outputs.Outputs.Bit15
          output Application.GPIO_HANDLER.IN_8 : BOOL  // Outputs.Outputs.Bit0
          output Application.GPIO_HANDLER.IN_9 : BOOL  // Outputs.Outputs.Bit1
          output Application.GPIO_HANDLER.IN_10 : BOOL  // Outputs.Outputs.Bit2
          output Application.GPIO_HANDLER.IN_11 : BOOL  // Outputs.Outputs.Bit3
          output Application.PLC_PRG.climate_state_reg : WORD  // Outputs.Outputs
          output Application.PLC_PRG.climate_temp_in : WORD  // Outputs.Outputs
          output Application.PLC_PRG.climate_temp_out : WORD  // Outputs.Outputs
          unmapped channels: Inputs, Outputs
  text list GlobalTextList
  5ce3da45-db07-42e7-a21c-a00fff4ed8f6|Images\bg_800.png
  5ce3da45-db07-42e7-a21c-a00fff4ed8f6|Images\mpx_state_bg.png
  5ce3da45-db07-42e7-a21c-a00fff4ed8f6|Images\ups\bypass_line_on.png
  5ce3da45-db07-42e7-a21c-a00fff4ed8f6|Images\ups\bypass_line_off.png
  5ce3da45-db07-42e7-a21c-a00fff4ed8f6|Images\ups\battery_arrow_off.png
  5ce3da45-db07-42e7-a21c-a00fff4ed8f6|Images\ups\battery_arrow_on.png
  5ce3da45-db07-42e7-a21c-a00fff4ed8f6|Images\ups\battery_line_off.png
  5ce3da45-db07-42e7-a21c-a00fff4ed8f6|Images\ups\battery_line_on.png
  5ce3da45-db07-42e7-a21c-a00fff4ed8f6|Images\ups\bypass_arrow_off.png
  5ce3da45-db07-42e7-a21c-a00fff4ed8f6|Images\ups\bypass_arrow_on.png
  5ce3da45-db07-42e7-a21c-a00fff4ed8f6|Images\ups\arrow_off.png
  5ce3da45-db07-42e7-a21c-a00fff4ed8f6|Images\ups\arrow_on.png
  5ce3da45-db07-42e7-a21c-a00fff4ed8f6|C:\workspace\SmiuUGP\Images\Proba.png
  5ce3da45-db07-42e7-a21c-a00fff4ed8f6|C:\workspace\SmiuUGP\Images\main_bg.png
  5ce3da45-db07-42e7-a21c-a00fff4ed8f6|C:\workspace\SmiuUGP\Images\bg_800.png
  5ce3da45-db07-42e7-a21c-a00fff4ed8f6|E:\YandexDisk\Скриншоты\ups.png
  5ce3da45-db07-42e7-a21c-a00fff4ed8f6|C:\workspace\SmiuUGP\Images\mpx_state_bg.png
  5ce3da45-db07-42e7-a21c-a00fff4ed8f6|C:\workspace\SmiuUGP\Images\scheme.png
  5ce3da45-db07-42e7-a21c-a00fff4ed8f6|C:\workspace\SmiuUGP\Images\more_info.png
  5ce3da45-db07-42e7-a21c-a00fff4ed8f6|C:\workspace\SmiuUGP\Images\log.png
  5ce3da45-db07-42e7-a21c-a00fff4ed8f6|C:\workspace\SmiuUGP\Images\gpio_1.png
  5ce3da45-db07-42e7-a21c-a00fff4ed8f6|C:\workspace\SmiuUGP\Images\schrpa.png
  5ce3da45-db07-42e7-a21c-a00fff4ed8f6|C:\workspace\SmiuUGP\Images\volt.png
  5ce3da45-db07-42e7-a21c-a00fff4ed8f6|C:\workspace\SmiuUGP\Images\shasn.png
  5ce3da45-db07-42e7-a21c-a00fff4ed8f6|C:\workspace\SmiuUGP\Images\schrps.png
  5ce3da45-db07-42e7-a21c-a00fff4ed8f6|C:\workspace\SmiuUGP\Images\battery.png
  5ce3da45-db07-42e7-a21c-a00fff4ed8f6|C:\workspace\SmiuUGP\Images\climate.png
  5ce3da45-db07-42e7-a21c-a00fff4ed8f6|C:\workspace\SmiuUGP\Images\alert.png
  5ce3da45-db07-42e7-a21c-a00fff4ed8f6|C:\workspace\SmiuUGP\Images\automation.png
  5ce3da45-db07-42e7-a21c-a00fff4ed8f6|E:\SmiuLinux\smiu_logo.png
  5ce3da45-db07-42e7-a21c-a00fff4ed8f6|C:\workspace\SmiuUGP\Images\mini_ups.png
*)

// CODESYS_Control_for_Raspberry_Pi/Application/PLC_PRG
PROGRAM PLC_PRG
VAR	

	//Тестовая плата
	pot_1 : WORD;
	pot_2 : WORD;
	pot_3 : WORD;

	//Визуализация
	var_true :BOOL := TRUE;
	ack		 :BOOL;
	history  :BOOL;	
	
	//Переменные для работы с МВ110-16 (адрес = 2)
	mv110_reg	                   :WORD; //Регистр состояния входов МВ110-16
	mv110_reg_as_bit 	           :WORD_AS_BIT; 
	mv110_in_0_in_main_present 	   :BOOL; //ШАСН - Наличие напряжения на основном вводе
	mv110_in_1_in_reserve_present  :BOOL; //ШАСН - Наличие напряжения на резервном вводе
	mv110_in_2_bp_sn_present 	   :BOOL; //ШАСН - Наличиче напряжения на БП СН
	mv110_in_3_gp_sn_present       :BOOL; //ШАСН - Наличие напряжения на ГП СН
	mv110_in_4_qs1_1position       :BOOL; //ШАСН - QS1 в первом положении
	mv110_in_5_qs1_2position       :BOOL; //ШАСН - QS1 во втором положении
	mv110_in_6_heat_on             :BOOL; //Обогрев включен
	mv110_in_7_gp1_u_fault 	       :BOOL; //ЩРПС - Исчезновение напряжения на ГП1
	mv110_in_8_gp2_u_fault 	       :BOOL; //ЩРПС - Исчезновение напряжения на ГП2
	
	//GPIO
	in_1_alarm_shos       :BOOL; //Нарушение ШОС IN_1
	in_2_alarm_fire       :BOOL; //Пожар IN_2
	in_3_alarm_shos_fault :BOOL; //Неисправность ШОС IN_3
	in_4_input_1_present  :BOOL; //ЩРПА: Наличие напряжения на 1 вводе IN_4
	in_5_input_2_present  :BOOL; //ЩРПА: Наличие напряжения на 2 вводе IN_5
	in_6_qs_1_pos_1       :BOOL; //ЩРПА: QS1 в первом положении IN_6
	in_7_qs_1_pos_2       :BOOL; //ЩРПА: QS1 во втором положении IN_7
	in_8_qs_2_pos_1       :BOOL; //ЩРПА: QS2 в первом положении IN_8
	in_9_qs_2_pos_2       :BOOL; //ЩРПА: QS2 во втором положении IN_9
	in_10_qs_3_pos_1      :BOOL; //ЩРПА: QS3 в первом положении IN_10
	in_11_qs_3_pos_2      :BOOL; //ЩРПА: QS3 во втором положении IN_11
	
	//Переменные для работы с климатом
	climate_temp_out          :WORD; 
	climat_temp_out_minus     :BOOL; //Бит отрицательности температуры
	climate_temp_out_real     :REAL; //Наружная температура
	climate_temp_in           :WORD; 
	climat_temp_in_minus      :BOOL; //Бит отрицательности температуры
	climate_temp_in_real      :REAL; //Внутренняя температура
	climate_state_reg         :WORD; 
	climate_state_as_bit      :WORD_AS_BIT;
	climate_zaslonka_state    :BOOL; //Состояние заслонки
	climate_vent_1_state      :BOOL; //Состояние вентилятора №1
	climate_vent_2_state      :BOOL; //Состояние вентилятора №2
	climate_condition_1_state :BOOL; //Состояние кондиционера №1
	climate_condition_2_state :BOOL; //Состояние кондиционера №2
	climate_heat_state        :BOOL; //Состояние обогрева
	climate_heat_door_state   :BOOL; //Состояние обогрева дверей
	climate_auto_state        :BOOL; //Состояние автоматики климата
	climate_temp_excess       :BOOL; //авария. внутренняя температура > 25
	
	//Переменные для работы с MPX_a1_1
	mpx_a1_1_in_v_1 	 		   		:WORD; //1-е Напрядение входа
	mpx_a1_1_in_v_2 	 		   		:WORD; //2-e Напряжение входа
	mpx_a1_1_in_v_3 	 		   		:WORD; //3-е Напряжение входа
	mpx_a1_1_in_freq 	 		   		:WORD; //Частота на входе
	mpx_a1_1_in_freq_real		   		:REAL; //Частота на входе (x0.1)
	mpx_a1_1_bypass_v_1  		   		:WORD; //1-е Напряжение байпаса
	mpx_a1_1_bypass_freq 		   		:WORD; //Частота байпаса
	mpx_a1_1_bypass_freq_real      		:REAL; //Частота байпаса
	mpx_a1_1_output_v_1  		   		:WORD; //1-е Напряжение выхода
	mpx_a1_1_output_i_1  		   		:WORD; //1-й Ток выхода
	mpx_a1_1_output_i_1_real       		:REAL; //1-й Ток выхода (x0.1)
	mpx_a1_1_output_active_power_1 		:WORD; //Активная мощность 1-й фазы
	mpx_a1_1_output_active_power_1_real :REAL; //Активная мощность 1-й фазы (x0.1)
	mpx_a1_1_output_freq 	       		:WORD; //Частота выхода
	mpx_a1_1_output_freq_real 	        :REAL; //Частота выхода (x0.1)
	mpx_a1_1_load_ph_1    	       		:WORD; //Загрузска 1-й фазы (%)
	mpx_a1_1_battery_voltage 	   		:WORD; //Напряжение батареи
	mpx_a1_1_battery_voltage_real  		:REAL; //Напряжение батареи (x0.1)
	mpx_a1_1_battery_current 	   		:WORD; //Ток батареи
	mpx_a1_1_battery_current_real  		:REAL; //Ток батареи (x0.1)
	mpx_a1_1_battery_capacity 	   		:WORD; //Остаточная емкость батареи (%)
	mpx_a1_1_battery_time 		   		:WORD; //Остаточное время автономии (минуты)
	mpx_a1_1_temp 				   		:WORD; //Температура
	mpx_a1_1_state_reg_1 	       		:WORD; //1-й Регистр состояния
	mpx_a1_1_state_1_as_bit 	   		:WORD_AS_BIT;
	mpx_a1_1_state_reg_2 		   		:WORD; //2-й Регистр состояния
	mpx_a1_1_state_2_as_bit 	   		:WORD_AS_BIT;
	mpx_a1_1_bypass_line_state 	   		:STRING; 
	mpx_a1_1_bypass_arrow_state    		:STRING;
	mpx_a1_1_battery_arrow_state 		:STRING; //состояние батареи
	mpx_a1_1_battery_line_state 		:STRING; //состояние батареи
	mpx_a1_1_input_state 		   		:STRING; //состояние входа
	mpx_a1_1_output_state 		   		:STRING; //состояние выхода
	mpx_a1_1_alarm                      :BOOL;
	
	//Переменные для работы с MPX_a1_2
	mpx_a1_2_in_v_1 	 		   		:WORD; //1-е Напрядение входа
	mpx_a1_2_in_v_2 	 		   		:WORD; //2-e Напряжение входа
	mpx_a1_2_in_v_3 	 		   		:WORD; //3-е Напряжение входа
	mpx_a1_2_in_freq 	 		   		:WORD; //Частота на входе
	mpx_a1_2_in_freq_real		   		:REAL; //Частота на входе (x0.1)
	mpx_a1_2_bypass_v_1  		   		:WORD; //1-е Напряжение байпаса
	mpx_a1_2_bypass_v_2  		   		:WORD; //2-е Напряжение байпаса
	mpx_a1_2_bypass_v_3  		   		:WORD; //3-е Напряжение байпаса
	mpx_a1_2_bypass_freq 		   		:WORD; //Частота байпаса
	mpx_a1_2_bypass_freq_real      		:REAL; //Частота байпаса
	mpx_a1_2_output_v_1  		   		:WORD; //1-е Напряжение выхода
	mpx_a1_2_output_v_2  		   		:WORD; //2-е Напряжение выхода
	mpx_a1_2_output_v_3  		   		:WORD; //3-е Напряжение выхода
	mpx_a1_2_output_i_1  		   		:WORD; //1-й Ток выхода
	mpx_a1_2_output_i_2  		   		:WORD; //2-й Ток выхода
	mpx_a1_2_output_i_3  		   		:WORD; //3-й Ток выхода
	mpx_a1_2_output_i_1_real       		:REAL; //1-й Ток выхода (x0.1)
	mpx_a1_2_output_i_2_real       		:REAL; //2-й Ток выхода (x0.1)
	mpx_a1_2_output_i_3_real       		:REAL; //3-й Ток выхода (x0.1)
	mpx_a1_2_output_active_power_1 		:WORD; //Активная мощность 1-й фазы
	mpx_a1_2_output_active_power_2 		:WORD; //Активная мощность 2-й фазы
	mpx_a1_2_output_active_power_3 		:WORD; //Активная мощность 3-й фазы
	mpx_a1_2_output_active_power_1_real :REAL; //Активная мощность 1-й фазы (x0.1)
	mpx_a1_2_output_active_power_2_real :REAL; //Активная мощность 2-й фазы (x0.1)
	mpx_a1_2_output_active_power_3_real :REAL; //Активная мощность 3-й фазы (x0.1)
	mpx_a1_2_output_freq 	       		:WORD; //Частота выхода
	mpx_a1_2_output_freq_real 	        :REAL; //Частота выхода (x0.1)
	mpx_a1_2_load_ph_1    	       		:WORD; //Загрузска 1-й фазы (%)
	mpx_a1_2_load_ph_2    		   		:WORD; //Загрузска 3-й фазы (%)
	mpx_a1_2_load_ph_3    	       		:WORD; //Загрузска 2-й фазы (%)
	mpx_a1_2_battery_voltage 	   		:WORD; //Напряжение батареи
	mpx_a1_2_battery_voltage_real  		:REAL; //Напряжение батареи (x0.1)
	mpx_a1_2_battery_current 	   		:WORD; //Ток батареи
	mpx_a1_2_battery_current_real  		:REAL; //Ток батареи (x0.1)
	mpx_a1_2_battery_capacity 	   		:WORD; //Остаточная емкость батареи (%)
	mpx_a1_2_battery_time 		   		:WORD; //Остаточное время автономии (минуты)
	mpx_a1_2_temp 				   		:WORD; //Температура
	mpx_a1_2_state_reg_1 	       		:WORD; //1-й Регистр состояния
	mpx_a1_2_state_1_as_bit 	   		:WORD_AS_BIT;
	mpx_a1_2_state_reg_2 		   		:WORD; //2-й Регистр состояния
	mpx_a1_2_state_2_as_bit 	   		:WORD_AS_BIT;
	mpx_a1_2_bypass_line_state 	   		:STRING; 
	mpx_a1_2_bypass_arrow_state    		:STRING;
	mpx_a1_2_battery_arrow_state 		:STRING; //состояние батареи
	mpx_a1_2_battery_line_state 		:STRING; //состояние батареи
	mpx_a1_2_input_state 		   		:STRING; //состояние входа
	mpx_a1_2_output_state 		   		:STRING; //состояние выхода
	mpx_a1_2_alarm                      :BOOL;
	
		//Переменные для работы с MPX_a2_1
	mpx_a2_1_in_v_1 	 		   		:WORD; //1-е Напрядение входа
	mpx_a2_1_in_v_2 	 		   		:WORD; //2-e Напряжение входа
	mpx_a2_1_in_v_3 	 		   		:WORD; //3-е Напряжение входа
	mpx_a2_1_in_freq 	 		   		:WORD; //Частота на входе
	mpx_a2_1_in_freq_real		   		:REAL; //Частота на входе (x0.1)
	mpx_a2_1_bypass_v_1  		   		:WORD; //1-е Напряжение байпаса
	mpx_a2_1_bypass_v_2  		   		:WORD; //2-е Напряжение байпаса
	mpx_a2_1_bypass_v_3  		   		:WORD; //3-е Напряжение байпаса
	mpx_a2_1_bypass_freq 		   		:WORD; //Частота байпаса
	mpx_a2_1_bypass_freq_real      		:REAL; //Частота байпаса
	mpx_a2_1_output_v_1  		   		:WORD; //1-е Напряжение выхода
	mpx_a2_1_output_v_2  		   		:WORD; //2-е Напряжение выхода
	mpx_a2_1_output_v_3  		   		:WORD; //3-е Напряжение выхода
	mpx_a2_1_output_i_1  		   		:WORD; //1-й Ток выхода
	mpx_a2_1_output_i_2  		   		:WORD; //2-й Ток выхода
	mpx_a2_1_output_i_3  		   		:WORD; //3-й Ток выхода
	mpx_a2_1_output_i_1_real       		:REAL; //1-й Ток выхода (x0.1)
	mpx_a2_1_output_i_2_real       		:REAL; //2-й Ток выхода (x0.1)
	mpx_a2_1_output_i_3_real       		:REAL; //3-й Ток выхода (x0.1)
	mpx_a2_1_output_active_power_1 		:WORD; //Активная мощность 1-й фазы
	mpx_a2_1_output_active_power_2 		:WORD; //Активная мощность 2-й фазы
	mpx_a2_1_output_active_power_3 		:WORD; //Активная мощность 3-й фазы
	mpx_a2_1_output_active_power_1_real :REAL; //Активная мощность 1-й фазы (x0.1)
	mpx_a2_1_output_active_power_2_real :REAL; //Активная мощность 2-й фазы (x0.1)
	mpx_a2_1_output_active_power_3_real :REAL; //Активная мощность 3-й фазы (x0.1)
	mpx_a2_1_output_freq 	       		:WORD; //Частота выхода
	mpx_a2_1_output_freq_real 	        :REAL; //Частота выхода (x0.1)
	mpx_a2_1_load_ph_1    	       		:WORD; //Загрузска 1-й фазы (%)
	mpx_a2_1_load_ph_2    		   		:WORD; //Загрузска 3-й фазы (%)
	mpx_a2_1_load_ph_3    	       		:WORD; //Загрузска 2-й фазы (%)
	mpx_a2_1_battery_voltage 	   		:WORD; //Напряжение батареи
	mpx_a2_1_battery_voltage_real  		:REAL; //Напряжение батареи (x0.1)
	mpx_a2_1_battery_current 	   		:WORD; //Ток батареи
	mpx_a2_1_battery_current_real  		:REAL; //Ток батареи (x0.1)
	mpx_a2_1_battery_capacity 	   		:WORD; //Остаточная емкость батареи (%)
	mpx_a2_1_battery_time 		   		:WORD; //Остаточное время автономии (минуты)
	mpx_a2_1_temp 				   		:WORD; //Температура
	mpx_a2_1_state_reg_1 	       		:WORD; //1-й Регистр состояния
	mpx_a2_1_state_1_as_bit 	   		:WORD_AS_BIT;
	mpx_a2_1_state_reg_2 		   		:WORD; //2-й Регистр состояния
	mpx_a2_1_state_2_as_bit 	   		:WORD_AS_BIT;
	mpx_a2_1_bypass_line_state 	   		:STRING; 
	mpx_a2_1_bypass_arrow_state    		:STRING;
	mpx_a2_1_battery_arrow_state 		:STRING; //состояние батареи
	mpx_a2_1_battery_line_state 		:STRING; //состояние батареи
	mpx_a2_1_input_state 		   		:STRING; //состояние входа
	mpx_a2_1_output_state 		   		:STRING; //состояние выхода
	mpx_a2_1_alarm                      :BOOL;
	
